// SIMATIC STEP 7 (V5.x) project CDCX52_Cordoba
// CPU: CPU
// station: P_ADR_BUS
// station: _S7H_BUSSYSTEM_CT
// station: Matériel
// station: API
// station: P_ADR_BUS
// station: Configuration
// station: MOP
// program: PROG
// program: Programa S7_BACK

SYMBOL_TABLE
"IBD"	DB 95	DB 95	// FACILITY: DATA BASE DB / DB BASE DE DONNEE
"IIT"	DB 96	DB 96	// FACILITY: PART TABLE / DB TABLE PIECE
"IIS"	DB 97	DB 97	// FACILITY: SUPPORT WORD TABLE / DB MOTS SUPPORT
"IG"	DB 99	DB 99	// FACILITY: GLOBAL DB / DB GLOBAL
END_SYMBOL_TABLE

DATA_BLOCK "IBD"	// DB 95
TITLE = FACILITY: DATABASE DB CONTROL
NAME : IBD
VERSION : 0.1
  STRUCT
   BDD : ARRAY  [1 .. 6, 1 .. 210 ] OF WORD ;	//SPARE
  END_STRUCT ;	
BEGIN
END_DATA_BLOCK

DATA_BLOCK "IIT"	// DB 96
TITLE = FACILITY: PART WORD TABLE
NAME : IIT
VERSION : 1.0
  STRUCT
   A01 : STRUCT 	//PALABRA PIEZA A01
    MP : STRUCT 	//PART MEMORY / PALABRA PIEZA
     MPP : BOOL ;	//PRESENT PART MEMORY / MEMORIA PIEZA PRESENTE
     MPAT : BOOL ;	//PART WITH WORK MEMORY / MEMORIA PIEZA A TRABAJAR
     MPST : BOOL ;	//PART WITHOUT WORK MEMORY / MEMORIA PIEZA SIN TRABAJO
     MPAM : BOOL ;	//PART MEMORY TO MATCH / MEMORIA PIEZA A CASAR
     MPAE : BOOL ;	//PART MEMORY TO EVACUATE / MEMORIA PIEZA A EVACUAR
     MPP1 : BOOL ;	//INTERMEDIATE PRESENT PART MEMORY / MEMORIA PIEZA PRESENTE INTERMEDIA
     MPP2 : BOOL ;	//INTERMEDIATE PRESENT PART MEMORY / MEMORIA PIEZA PRESENTE INTERMEDIA
     MPP3 : BOOL ;	//INTERMEDIATE PRESENT PART MEMORY / MEMORIA PIEZA PRESENTE INTERMEDIA
     MPP4 : BOOL ;	//INTERMEDIATE PRESENT PART MEMORY / MEMORIA PIEZA PRESENTE INTERMEDIA
     MPP5 : BOOL ;	//INTERMEDIATE PRESENT PART MEMORY / MEMORIA PIEZA PRESENTE INTERMEDIA
     MPP6 : BOOL ;	//INTERMEDIATE PRESENT PART MEMORY / MEMORIA PIEZA PRESENTE INTERMEDIA
     MPP7 : BOOL ;	//INTERMEDIATE PRESENT PART MEMORY / MEMORIA PIEZA PRESENTE INTERMEDIA
     MPP8 : BOOL ;	//INTERMEDIATE PRESENT PART MEMORY / MEMORIA PIEZA PRESENTE INTERMEDIA
     MPT : BOOL ;	//PART COMPLETE MEMORY / MEMORIA PIEZA TRABAJADA
     MPLNOK : BOOL ;	//LAUCHING PART MEMORY NOK / MEMORIA LANZAMIENTO PIEZA NO OK
     MPLNOR : BOOL ;	//LAUCHING PART MEMORY OK / MEMORIA LANZAMIENTO PIEZA OK
    END_STRUCT ;
    MS : INT ;
    NFILM : INT ;	//FILM NUMBER / NUMERO DE FILMO
    NORDRE : INT ;	//ORDER NUMBER / NUMERO DE ORDEN
    CDIV1 : INT ;	//FAMILIA (CDIV1)
    CDIV2 : INT ;	//FASE (CDIV2)
    CDIV3 : INT ;	//MODELO (CDIV3)
    CDIV4 : INT ;	//TECHO (CDIV4)
    CDIV5 : INT ;	//VERSION (CDIV5)
    DESFI : INT ;	//FINAL DISPATCH / DESTINO FINAL
    CSORT : INT ;	//TRADUCTION / CAUSA DE SALIDA
    DAT : STRUCT 	//DEFINICION / ESPERA TRABAJO
     B8 : BOOL ;
     B9 : BOOL ;
     B10 : BOOL ;
     B11 : BOOL ;
     B12 : BOOL ;
     FABSPF : BOOL ;	//FABRICACION SIN PIEZA AL FILMO
     B14 : BOOL ;
     B15 : BOOL ;
     B0 : BOOL ;
     B1 : BOOL ;
     B2 : BOOL ;
     B3 : BOOL ;
     B4 : BOOL ;
     B5 : BOOL ;
     B6 : BOOL ;
     B7 : BOOL ;
    END_STRUCT ;
    CRAPI : STRUCT 	//PLC DISPATCHING REASON / CAUSA ENRUTADO API
     B8 : BOOL ;
     B9 : BOOL ;
     B10 : BOOL ;
     B11 : BOOL ;
     B12 : BOOL ;
     B13 : BOOL ;
     B14 : BOOL ;
     B15 : BOOL ;
     B0 : BOOL ;
     B1 : BOOL ;
     B2 : BOOL ;
     RARET : BOOL ;	//PIEZA ANALISIS - RETOQUE
     B4 : BOOL ;
     B5 : BOOL ;
     B6 : BOOL ;
     B7 : BOOL ;
    END_STRUCT ;
    MGEST : STRUCT 	//PALABRA DE GESTION RECALAJE
     MPFNOR : BOOL ;	//MEMORIA PIEZA FLUJO NORMAL
     MPSTC : BOOL ;	//MEMORIA PIEZA A SALIR TODOS LOS CASOS
     MPSOR : BOOL ;	//MEMORIA PIEZA A SALIR (SALIDA SIPTOL BUENA)
     MPSSU : BOOL ;	//MEMORIA PIEZA A SALIR (SUSTITUCION PIEZA BUENA)
     MPSDI : BOOL ;	//MEMORIA PIEZA A SALIR (DISCORDANCIA)
     MPSSUL : BOOL ;	//MEMORIA PIEZA A SALIR (SUSTITUCION PIEZA MALA)
     MPSL : BOOL ;	//MEMORIA PIEZA A SALIR (SALIDA MALA)
     MPSF99 : BOOL ;	//MEMORIA PIEZA A SALIR (MAP FILM 99)
     MPETC : BOOL ;	//MEMORIA PIEZA A ENTRAR TODOS LOS CASOS
     MPEOR : BOOL ;	//MEMORIA PIEZA EN ENTRADA (DEMANDA SIPTOL)
     MPESUB : BOOL ;	//MEMORIA PIEZA EN ENTRADA (SUSTITUCION PIEZA BUENA)
     MPEDI : BOOL ;	//MEMORIA PIEZA EN ENTRADA (DISCORDANCIA)
     MPESUL : BOOL ;	//MEMORIA PIEZA EN ENTRADA (SUSTITUCION PIEZA MALA)
     MPOCV : BOOL ;	//MEMORIA PIEZA A SALIR VEHICULO ANULADO + GANCHO VACIO
     MESUTC : BOOL ;	//MEMORIA EN ENTRADA SUSTITUCION TODOS LOS CASOS (PIEZA BUENA O MALA)
     MSSUTC : BOOL ;	//MEMORIA SALIDA SUSTITUCION TODOS LOS CASOS (PIEZA BUENA O MALA)
    END_STRUCT ;
    TVEH : STRUCT 	//TYPO DE VEHICULO
     B8 : BOOL ;
     B9 : BOOL ;
     B10 : BOOL ;
     B11 : BOOL ;
     B12 : BOOL ;
     B13 : BOOL ;
     B14 : BOOL ;
     FABSPF : BOOL ;	//FABRICACION SIN PIEZA AL FILMO
     SPE : BOOL ;	//UNIT ESPECIAL
     B1 : BOOL ;
     B2 : BOOL ;
     B3 : BOOL ;
     B4 : BOOL ;
     B5 : BOOL ;
     B6 : BOOL ;
     B7 : BOOL ;
    END_STRUCT ;
    SPARE : ARRAY  [1 .. 5 ] OF INT ;	//SPARE
   END_STRUCT ;
   B01 : STRUCT 	//PALABRA PIEZA B01
    MP : STRUCT 	//PART MEMORY / PALABRA PIEZA
     MPP : BOOL ;	//PRESENT PART MEMORY / MEMORIA PIEZA PRESENTE
     MPAT : BOOL ;	//PART WITH WORK MEMORY / MEMORIA PIEZA A TRABAJAR
     MPST : BOOL ;	//PART WITHOUT WORK MEMORY / MEMORIA PIEZA SIN TRABAJO
     MPAM : BOOL ;	//PART MEMORY TO MATCH / MEMORIA PIEZA A CASAR
     MPAE : BOOL ;	//PART MEMORY TO EVACUATE / MEMORIA PIEZA A EVACUAR
     MPP1 : BOOL ;	//INTERMEDIATE PRESENT PART MEMORY / MEMORIA PIEZA PRESENTE INTERMEDIA
     MPP2 : BOOL ;	//INTERMEDIATE PRESENT PART MEMORY / MEMORIA PIEZA PRESENTE INTERMEDIA
     MPP3 : BOOL ;	//INTERMEDIATE PRESENT PART MEMORY / MEMORIA PIEZA PRESENTE INTERMEDIA
     MPP4 : BOOL ;	//INTERMEDIATE PRESENT PART MEMORY / MEMORIA PIEZA PRESENTE INTERMEDIA
     MPP5 : BOOL ;	//INTERMEDIATE PRESENT PART MEMORY / MEMORIA PIEZA PRESENTE INTERMEDIA
     MPP6 : BOOL ;	//INTERMEDIATE PRESENT PART MEMORY / MEMORIA PIEZA PRESENTE INTERMEDIA
     MPP7 : BOOL ;	//INTERMEDIATE PRESENT PART MEMORY / MEMORIA PIEZA PRESENTE INTERMEDIA
     MPP8 : BOOL ;	//INTERMEDIATE PRESENT PART MEMORY / MEMORIA PIEZA PRESENTE INTERMEDIA
     MPT : BOOL ;	//PART COMPLETE MEMORY / MEMORIA PIEZA TRABAJADA
     MPLNOK : BOOL ;	//LAUCHING PART MEMORY NOK / MEMORIA LANZAMIENTO PIEZA NO OK
     MPLNOR : BOOL ;	//LAUCHING PART MEMORY OK / MEMORIA LANZAMIENTO PIEZA OK
    END_STRUCT ;
    MS : INT ;
    NFILM : INT ;	//FILM NUMBER / NUMERO DE FILMO
    NORDRE : INT ;	//ORDER NUMBER / NUMERO DE ORDEN
    CDIV1 : INT ;	//FAMILIA (CDIV1)
    CDIV2 : INT ;	//FASE (CDIV2)
    CDIV3 : INT ;	//MODELO (CDIV3)
    CDIV4 : INT ;	//TECHO (CDIV4)
    CDIV5 : INT ;	//VERSION (CDIV5)
    DESFI : INT ;	//FINAL DISPATCH / DESTINO FINAL
    CSORT : INT ;	//TRADUCTION / CAUSA DE SALIDA
    DAT : STRUCT 	//DEFINICION / ESPERA TRABAJO
     B8 : BOOL ;
     B9 : BOOL ;
     B10 : BOOL ;
     B11 : BOOL ;
     B12 : BOOL ;
     FABSPF : BOOL ;	//FABRICACION SIN PIEZA AL FILMO
     B14 : BOOL ;
     B15 : BOOL ;
     B0 : BOOL ;
     B1 : BOOL ;
     B2 : BOOL ;
     B3 : BOOL ;
     B4 : BOOL ;
     B5 : BOOL ;
     B6 : BOOL ;
     B7 : BOOL ;
    END_STRUCT ;
    CRAPI : STRUCT 	//PLC DISPATCHING REASON / CAUSA ENRUTADO API
     B8 : BOOL ;
     B9 : BOOL ;
     B10 : BOOL ;
     B11 : BOOL ;
     B12 : BOOL ;
     B13 : BOOL ;
     B14 : BOOL ;
     B15 : BOOL ;
     B0 : BOOL ;
     B1 : BOOL ;
     B2 : BOOL ;
     RARET : BOOL ;	//PIEZA ANALISIS - RETOQUE
     B4 : BOOL ;
     B5 : BOOL ;
     B6 : BOOL ;
     B7 : BOOL ;
    END_STRUCT ;
    MGEST : STRUCT 	//PALABRA DE GESTION RECALAJE
     MPFNOR : BOOL ;	//MEMORIA PIEZA FLUJO NORMAL
     MPSTC : BOOL ;	//MEMORIA PIEZA A SALIR TODOS LOS CASOS
     MPSOR : BOOL ;	//MEMORIA PIEZA A SALIR (SALIDA SIPTOL BUENA)
     MPSSU : BOOL ;	//MEMORIA PIEZA A SALIR (SUSTITUCION PIEZA BUENA)
     MPSDI : BOOL ;	//MEMORIA PIEZA A SALIR (DISCORDANCIA)
     MPSSUL : BOOL ;	//MEMORIA PIEZA A SALIR (SUSTITUCION PIEZA MALA)
     MPSL : BOOL ;	//MEMORIA PIEZA A SALIR (SALIDA MALA)
     MPSF99 : BOOL ;	//MEMORIA PIEZA A SALIR (MAP FILM 99)
     MPETC : BOOL ;	//MEMORIA PIEZA A ENTRAR TODOS LOS CASOS
     MPEOR : BOOL ;	//MEMORIA PIEZA EN ENTRADA (DEMANDA SIPTOL)
     MPESUB : BOOL ;	//MEMORIA PIEZA EN ENTRADA (SUSTITUCION PIEZA BUENA)
     MPEDI : BOOL ;	//MEMORIA PIEZA EN ENTRADA (DISCORDANCIA)
     MPESUL : BOOL ;	//MEMORIA PIEZA EN ENTRADA (SUSTITUCION PIEZA MALA)
     MPOCV : BOOL ;	//MEMORIA PIEZA A SALIR VEHICULO ANULADO + GANCHO VACIO
     MESUTC : BOOL ;	//MEMORIA EN ENTRADA SUSTITUCION TODOS LOS CASOS (PIEZA BUENA O MALA)
     MSSUTC : BOOL ;	//MEMORIA SALIDA SUSTITUCION TODOS LOS CASOS (PIEZA BUENA O MALA)
    END_STRUCT ;
    TVEH : STRUCT 	//TYPO DE VEHICULO
     B8 : BOOL ;
     B9 : BOOL ;
     B10 : BOOL ;
     B11 : BOOL ;
     B12 : BOOL ;
     B13 : BOOL ;
     B14 : BOOL ;
     FABSPF : BOOL ;	//FABRICACION SIN PIEZA AL FILMO
     SPE : BOOL ;	//UNIT ESPECIAL
     B1 : BOOL ;
     B2 : BOOL ;
     B3 : BOOL ;
     B4 : BOOL ;
     B5 : BOOL ;
     B6 : BOOL ;
     B7 : BOOL ;
    END_STRUCT ;
    SPARE : ARRAY  [1 .. 5 ] OF INT ;
   END_STRUCT ;
   B02 : STRUCT 	//PALABRA PIEZA B02
    MP : STRUCT 	//PART MEMORY / PALABRA PIEZA
     MPP : BOOL ;	//PRESENT PART MEMORY / MEMORIA PIEZA PRESENTE
     MPAT : BOOL ;	//PART WITH WORK MEMORY / MEMORIA PIEZA A TRABAJAR
     MPST : BOOL ;	//PART WITHOUT WORK MEMORY / MEMORIA PIEZA SIN TRABAJO
     MPAM : BOOL ;	//PART MEMORY TO MATCH / MEMORIA PIEZA A CASAR
     MPAE : BOOL ;	//PART MEMORY TO EVACUATE / MEMORIA PIEZA A EVACUAR
     MPP1 : BOOL ;	//INTERMEDIATE PRESENT PART MEMORY / MEMORIA PIEZA PRESENTE INTERMEDIA
     MPP2 : BOOL ;	//INTERMEDIATE PRESENT PART MEMORY / MEMORIA PIEZA PRESENTE INTERMEDIA
     MPP3 : BOOL ;	//INTERMEDIATE PRESENT PART MEMORY / MEMORIA PIEZA PRESENTE INTERMEDIA
     MPP4 : BOOL ;	//INTERMEDIATE PRESENT PART MEMORY / MEMORIA PIEZA PRESENTE INTERMEDIA
     MPP5 : BOOL ;	//INTERMEDIATE PRESENT PART MEMORY / MEMORIA PIEZA PRESENTE INTERMEDIA
     MPP6 : BOOL ;	//INTERMEDIATE PRESENT PART MEMORY / MEMORIA PIEZA PRESENTE INTERMEDIA
     MPP7 : BOOL ;	//INTERMEDIATE PRESENT PART MEMORY / MEMORIA PIEZA PRESENTE INTERMEDIA
     MPP8 : BOOL ;	//INTERMEDIATE PRESENT PART MEMORY / MEMORIA PIEZA PRESENTE INTERMEDIA
     MPT : BOOL ;	//PART COMPLETE MEMORY / MEMORIA PIEZA TRABAJADA
     MPLNOK : BOOL ;	//LAUCHING PART MEMORY NOK / MEMORIA LANZAMIENTO PIEZA NO OK
     MPLNOR : BOOL ;	//LAUCHING PART MEMORY OK / MEMORIA LANZAMIENTO PIEZA OK
    END_STRUCT ;
    MS : INT ;
    NFILM : INT ;	//FILM NUMBER / NUMERO DE FILMO
    NORDRE : INT ;	//ORDER NUMBER / NUMERO DE ORDEN
    CDIV1 : INT ;	//FAMILIA (CDIV1)
    CDIV2 : INT ;	//FASE (CDIV2)
    CDIV3 : INT ;	//MODELO (CDIV3)
    CDIV4 : INT ;	//TECHO (CDIV4)
    CDIV5 : INT ;	//VERSION (CDIV5)
    DESFI : INT ;	//FINAL DISPATCH / DESTINO FINAL
    CSORT : INT ;	//TRADUCTION / CAUSA DE SALIDA
    DAT : STRUCT 	//DEFINICION / ESPERA TRABAJO
     B8 : BOOL ;
     B9 : BOOL ;
     B10 : BOOL ;
     B11 : BOOL ;
     B12 : BOOL ;
     FABSPF : BOOL ;	//FABRICACION SIN PIEZA AL FILMO
     B14 : BOOL ;
     B15 : BOOL ;
     B0 : BOOL ;
     B1 : BOOL ;
     B2 : BOOL ;
     B3 : BOOL ;
     B4 : BOOL ;
     B5 : BOOL ;
     B6 : BOOL ;
     B7 : BOOL ;
    END_STRUCT ;
    CRAPI : STRUCT 	//PLC DISPATCHING REASON / CAUSA ENRUTADO API
     B8 : BOOL ;
     B9 : BOOL ;
     B10 : BOOL ;
     B11 : BOOL ;
     B12 : BOOL ;
     B13 : BOOL ;
     B14 : BOOL ;
     B15 : BOOL ;
     B0 : BOOL ;
     B1 : BOOL ;
     B2 : BOOL ;
     RARET : BOOL ;	//PIEZA ANALISIS - RETOQUE
     B4 : BOOL ;
     B5 : BOOL ;
     B6 : BOOL ;
     B7 : BOOL ;
    END_STRUCT ;
    MGEST : STRUCT 	//PALABRA DE GESTION RECALAJE
     MPFNOR : BOOL ;	//MEMORIA PIEZA FLUJO NORMAL
     MPSTC : BOOL ;	//MEMORIA PIEZA A SALIR TODOS LOS CASOS
     MPSOR : BOOL ;	//MEMORIA PIEZA A SALIR (SALIDA SIPTOL BUENA)
     MPSSU : BOOL ;	//MEMORIA PIEZA A SALIR (SUSTITUCION PIEZA BUENA)
     MPSDI : BOOL ;	//MEMORIA PIEZA A SALIR (DISCORDANCIA)
     MPSSUL : BOOL ;	//MEMORIA PIEZA A SALIR (SUSTITUCION PIEZA MALA)
     MPSL : BOOL ;	//MEMORIA PIEZA A SALIR (SALIDA MALA)
     MPSF99 : BOOL ;	//MEMORIA PIEZA A SALIR (MAP FILM 99)
     MPETC : BOOL ;	//MEMORIA PIEZA A ENTRAR TODOS LOS CASOS
     MPEOR : BOOL ;	//MEMORIA PIEZA EN ENTRADA (DEMANDA SIPTOL)
     MPESUB : BOOL ;	//MEMORIA PIEZA EN ENTRADA (SUSTITUCION PIEZA BUENA)
     MPEDI : BOOL ;	//MEMORIA PIEZA EN ENTRADA (DISCORDANCIA)
     MPESUL : BOOL ;	//MEMORIA PIEZA EN ENTRADA (SUSTITUCION PIEZA MALA)
     MPOCV : BOOL ;	//MEMORIA PIEZA A SALIR VEHICULO ANULADO + GANCHO VACIO
     MESUTC : BOOL ;	//MEMORIA EN ENTRADA SUSTITUCION TODOS LOS CASOS (PIEZA BUENA O MALA)
     MSSUTC : BOOL ;	//MEMORIA SALIDA SUSTITUCION TODOS LOS CASOS (PIEZA BUENA O MALA)
    END_STRUCT ;
    TVEH : STRUCT 	//TYPO DE VEHICULO
     B8 : BOOL ;
     B9 : BOOL ;
     B10 : BOOL ;
     B11 : BOOL ;
     B12 : BOOL ;
     B13 : BOOL ;
     B14 : BOOL ;
     FABSPF : BOOL ;	//FABRICACION SIN PIEZA AL FILMO
     SPE : BOOL ;	//UNIT ESPECIAL
     B1 : BOOL ;
     B2 : BOOL ;
     B3 : BOOL ;
     B4 : BOOL ;
     B5 : BOOL ;
     B6 : BOOL ;
     B7 : BOOL ;
    END_STRUCT ;
    SPARE : ARRAY  [1 .. 5 ] OF INT ;
   END_STRUCT ;
   C01 : STRUCT 	//PALABRA PIEZA C01
    MP : STRUCT 	//PART MEMORY / PALABRA PIEZA
     MPP : BOOL ;	//PRESENT PART MEMORY / MEMORIA PIEZA PRESENTE
     MPAT : BOOL ;	//PART WITH WORK MEMORY / MEMORIA PIEZA A TRABAJAR
     MPST : BOOL ;	//PART WITHOUT WORK MEMORY / MEMORIA PIEZA SIN TRABAJO
     MPAM : BOOL ;	//PART MEMORY TO MATCH / MEMORIA PIEZA A CASAR
     MPAE : BOOL ;	//PART MEMORY TO EVACUATE / MEMORIA PIEZA A EVACUAR
     MPP1 : BOOL ;	//INTERMEDIATE PRESENT PART MEMORY / MEMORIA PIEZA PRESENTE INTERMEDIA
     MPP2 : BOOL ;	//INTERMEDIATE PRESENT PART MEMORY / MEMORIA PIEZA PRESENTE INTERMEDIA
     MPP3 : BOOL ;	//INTERMEDIATE PRESENT PART MEMORY / MEMORIA PIEZA PRESENTE INTERMEDIA
     MPP4 : BOOL ;	//INTERMEDIATE PRESENT PART MEMORY / MEMORIA PIEZA PRESENTE INTERMEDIA
     MPP5 : BOOL ;	//INTERMEDIATE PRESENT PART MEMORY / MEMORIA PIEZA PRESENTE INTERMEDIA
     MPP6 : BOOL ;	//INTERMEDIATE PRESENT PART MEMORY / MEMORIA PIEZA PRESENTE INTERMEDIA
     MPP7 : BOOL ;	//INTERMEDIATE PRESENT PART MEMORY / MEMORIA PIEZA PRESENTE INTERMEDIA
     MPP8 : BOOL ;	//INTERMEDIATE PRESENT PART MEMORY / MEMORIA PIEZA PRESENTE INTERMEDIA
     MPT : BOOL ;	//PART COMPLETE MEMORY / MEMORIA PIEZA TRABAJADA
     MPLNOK : BOOL ;	//LAUCHING PART MEMORY NOK / MEMORIA LANZAMIENTO PIEZA NO OK
     MPLNOR : BOOL ;	//LAUCHING PART MEMORY OK / MEMORIA LANZAMIENTO PIEZA OK
    END_STRUCT ;
    MS : INT ;
    NFILM : INT ;	//FILM NUMBER / NUMERO DE FILMO
    NORDRE : INT ;	//ORDER NUMBER / NUMERO DE ORDEN
    CDIV1 : INT ;	//FAMILIA (CDIV1)
    CDIV2 : INT ;	//FASE (CDIV2)
    CDIV3 : INT ;	//MODELO (CDIV3)
    CDIV4 : INT ;	//TECHO (CDIV4)
    CDIV5 : INT ;	//VERSION (CDIV5)
    DESFI : INT ;	//FINAL DISPATCH / DESTINO FINAL
    CSORT : INT ;	//TRADUCTION / CAUSA DE SALIDA
    DAT : STRUCT 	//DEFINICION / ESPERA TRABAJO
     B8 : BOOL ;
     B9 : BOOL ;
     B10 : BOOL ;
     B11 : BOOL ;
     B12 : BOOL ;
     FABSPF : BOOL ;	//FABRICACION SIN PIEZA AL FILMO
     B14 : BOOL ;
     B15 : BOOL ;
     B0 : BOOL ;
     B1 : BOOL ;
     B2 : BOOL ;
     B3 : BOOL ;
     B4 : BOOL ;
     B5 : BOOL ;
     B6 : BOOL ;
     B7 : BOOL ;
    END_STRUCT ;
    CRAPI : STRUCT 	//PLC DISPATCHING REASON / CAUSA ENRUTADO API
     B8 : BOOL ;
     B9 : BOOL ;
     B10 : BOOL ;
     B11 : BOOL ;
     B12 : BOOL ;
     B13 : BOOL ;
     B14 : BOOL ;
     B15 : BOOL ;
     B0 : BOOL ;
     B1 : BOOL ;
     B2 : BOOL ;
     RARET : BOOL ;	//PIEZA ANALISIS - RETOQUE
     B4 : BOOL ;
     B5 : BOOL ;
     B6 : BOOL ;
     B7 : BOOL ;
    END_STRUCT ;
    MGEST : STRUCT 	//PALABRA DE GESTION RECALAJE
     MPFNOR : BOOL ;	//MEMORIA PIEZA FLUJO NORMAL
     MPSTC : BOOL ;	//MEMORIA PIEZA A SALIR TODOS LOS CASOS
     MPSOR : BOOL ;	//MEMORIA PIEZA A SALIR (SALIDA SIPTOL BUENA)
     MPSSU : BOOL ;	//MEMORIA PIEZA A SALIR (SUSTITUCION PIEZA BUENA)
     MPSDI : BOOL ;	//MEMORIA PIEZA A SALIR (DISCORDANCIA)
     MPSSUL : BOOL ;	//MEMORIA PIEZA A SALIR (SUSTITUCION PIEZA MALA)
     MPSL : BOOL ;	//MEMORIA PIEZA A SALIR (SALIDA MALA)
     MPSF99 : BOOL ;	//MEMORIA PIEZA A SALIR (MAP FILM 99)
     MPETC : BOOL ;	//MEMORIA PIEZA A ENTRAR TODOS LOS CASOS
     MPEOR : BOOL ;	//MEMORIA PIEZA EN ENTRADA (DEMANDA SIPTOL)
     MPESUB : BOOL ;	//MEMORIA PIEZA EN ENTRADA (SUSTITUCION PIEZA BUENA)
     MPEDI : BOOL ;	//MEMORIA PIEZA EN ENTRADA (DISCORDANCIA)
     MPESUL : BOOL ;	//MEMORIA PIEZA EN ENTRADA (SUSTITUCION PIEZA MALA)
     MPOCV : BOOL ;	//MEMORIA PIEZA A SALIR VEHICULO ANULADO + GANCHO VACIO
     MESUTC : BOOL ;	//MEMORIA EN ENTRADA SUSTITUCION TODOS LOS CASOS (PIEZA BUENA O MALA)
     MSSUTC : BOOL ;	//MEMORIA SALIDA SUSTITUCION TODOS LOS CASOS (PIEZA BUENA O MALA)
    END_STRUCT ;
    TVEH : STRUCT 	//TYPO DE VEHICULO
     B8 : BOOL ;
     B9 : BOOL ;
     B10 : BOOL ;
     B11 : BOOL ;
     B12 : BOOL ;
     B13 : BOOL ;
     B14 : BOOL ;
     FABSPF : BOOL ;	//FABRICACION SIN PIEZA AL FILMO
     SPE : BOOL ;	//UNIT ESPECIAL
     B1 : BOOL ;
     B2 : BOOL ;
     B3 : BOOL ;
     B4 : BOOL ;
     B5 : BOOL ;
     B6 : BOOL ;
     B7 : BOOL ;
    END_STRUCT ;
    SPARE : ARRAY  [1 .. 5 ] OF INT ;
   END_STRUCT ;
   C02 : STRUCT 	//PALABRA PIEZA C02
    MP : STRUCT 	//PART MEMORY / PALABRA PIEZA
     MPP : BOOL ;	//PRESENT PART MEMORY / MEMORIA PIEZA PRESENTE
     MPAT : BOOL ;	//PART WITH WORK MEMORY / MEMORIA PIEZA A TRABAJAR
     MPST : BOOL ;	//PART WITHOUT WORK MEMORY / MEMORIA PIEZA SIN TRABAJO
     MPAM : BOOL ;	//PART MEMORY TO MATCH / MEMORIA PIEZA A CASAR
     MPAE : BOOL ;	//PART MEMORY TO EVACUATE / MEMORIA PIEZA A EVACUAR
     MPP1 : BOOL ;	//INTERMEDIATE PRESENT PART MEMORY / MEMORIA PIEZA PRESENTE INTERMEDIA
     MPP2 : BOOL ;	//INTERMEDIATE PRESENT PART MEMORY / MEMORIA PIEZA PRESENTE INTERMEDIA
     MPP3 : BOOL ;	//INTERMEDIATE PRESENT PART MEMORY / MEMORIA PIEZA PRESENTE INTERMEDIA
     MPP4 : BOOL ;	//INTERMEDIATE PRESENT PART MEMORY / MEMORIA PIEZA PRESENTE INTERMEDIA
     MPP5 : BOOL ;	//INTERMEDIATE PRESENT PART MEMORY / MEMORIA PIEZA PRESENTE INTERMEDIA
     MPP6 : BOOL ;	//INTERMEDIATE PRESENT PART MEMORY / MEMORIA PIEZA PRESENTE INTERMEDIA
     MPP7 : BOOL ;	//INTERMEDIATE PRESENT PART MEMORY / MEMORIA PIEZA PRESENTE INTERMEDIA
     MPP8 : BOOL ;	//INTERMEDIATE PRESENT PART MEMORY / MEMORIA PIEZA PRESENTE INTERMEDIA
     MPT : BOOL ;	//PART COMPLETE MEMORY / MEMORIA PIEZA TRABAJADA
     MPLNOK : BOOL ;	//LAUCHING PART MEMORY NOK / MEMORIA LANZAMIENTO PIEZA NO OK
     MPLNOR : BOOL ;	//LAUCHING PART MEMORY OK / MEMORIA LANZAMIENTO PIEZA OK
    END_STRUCT ;
    MS : INT ;
    NFILM : INT ;	//FILM NUMBER / NUMERO DE FILMO
    NORDRE : INT ;	//ORDER NUMBER / NUMERO DE ORDEN
    CDIV1 : INT ;	//FAMILIA (CDIV1)
    CDIV2 : INT ;	//FASE (CDIV2)
    CDIV3 : INT ;	//MODELO (CDIV3)
    CDIV4 : INT ;	//TECHO (CDIV4)
    CDIV5 : INT ;	//VERSION (CDIV5)
    DESFI : INT ;	//FINAL DISPATCH / DESTINO FINAL
    CSORT : INT ;	//TRADUCTION / CAUSA DE SALIDA
    DAT : STRUCT 	//DEFINICION / ESPERA TRABAJO
     B8 : BOOL ;
     B9 : BOOL ;
     B10 : BOOL ;
     B11 : BOOL ;
     B12 : BOOL ;
     FABSPF : BOOL ;	//FABRICACION SIN PIEZA AL FILMO
     B14 : BOOL ;
     B15 : BOOL ;
     B0 : BOOL ;
     B1 : BOOL ;
     B2 : BOOL ;
     B3 : BOOL ;
     B4 : BOOL ;
     B5 : BOOL ;
     B6 : BOOL ;
     B7 : BOOL ;
    END_STRUCT ;
    CRAPI : STRUCT 	//PLC DISPATCHING REASON / CAUSA ENRUTADO API
     B8 : BOOL ;
     B9 : BOOL ;
     B10 : BOOL ;
     B11 : BOOL ;
     B12 : BOOL ;
     B13 : BOOL ;
     B14 : BOOL ;
     B15 : BOOL ;
     B0 : BOOL ;
     B1 : BOOL ;
     B2 : BOOL ;
     RARET : BOOL ;	//PIEZA ANALISIS - RETOQUE
     B4 : BOOL ;
     B5 : BOOL ;
     B6 : BOOL ;
     B7 : BOOL ;
    END_STRUCT ;
    MGEST : STRUCT 	//PALABRA DE GESTION RECALAJE
     MPFNOR : BOOL ;	//MEMORIA PIEZA FLUJO NORMAL
     MPSTC : BOOL ;	//MEMORIA PIEZA A SALIR TODOS LOS CASOS
     MPSOR : BOOL ;	//MEMORIA PIEZA A SALIR (SALIDA SIPTOL BUENA)
     MPSSU : BOOL ;	//MEMORIA PIEZA A SALIR (SUSTITUCION PIEZA BUENA)
     MPSDI : BOOL ;	//MEMORIA PIEZA A SALIR (DISCORDANCIA)
     MPSSUL : BOOL ;	//MEMORIA PIEZA A SALIR (SUSTITUCION PIEZA MALA)
     MPSL : BOOL ;	//MEMORIA PIEZA A SALIR (SALIDA MALA)
     MPSF99 : BOOL ;	//MEMORIA PIEZA A SALIR (MAP FILM 99)
     MPETC : BOOL ;	//MEMORIA PIEZA A ENTRAR TODOS LOS CASOS
     MPEOR : BOOL ;	//MEMORIA PIEZA EN ENTRADA (DEMANDA SIPTOL)
     MPESUB : BOOL ;	//MEMORIA PIEZA EN ENTRADA (SUSTITUCION PIEZA BUENA)
     MPEDI : BOOL ;	//MEMORIA PIEZA EN ENTRADA (DISCORDANCIA)
     MPESUL : BOOL ;	//MEMORIA PIEZA EN ENTRADA (SUSTITUCION PIEZA MALA)
     MPOCV : BOOL ;	//MEMORIA PIEZA A SALIR VEHICULO ANULADO + GANCHO VACIO
     MESUTC : BOOL ;	//MEMORIA EN ENTRADA SUSTITUCION TODOS LOS CASOS (PIEZA BUENA O MALA)
     MSSUTC : BOOL ;	//MEMORIA SALIDA SUSTITUCION TODOS LOS CASOS (PIEZA BUENA O MALA)
    END_STRUCT ;
    TVEH : STRUCT 	//TYPO DE VEHICULO
     B8 : BOOL ;
     B9 : BOOL ;
     B10 : BOOL ;
     B11 : BOOL ;
     B12 : BOOL ;
     B13 : BOOL ;
     B14 : BOOL ;
     FABSPF : BOOL ;	//FABRICACION SIN PIEZA AL FILMO
     SPE : BOOL ;	//UNIT ESPECIAL
     B1 : BOOL ;
     B2 : BOOL ;
     B3 : BOOL ;
     B4 : BOOL ;
     B5 : BOOL ;
     B6 : BOOL ;
     B7 : BOOL ;
    END_STRUCT ;
    SPARE : ARRAY  [1 .. 5 ] OF INT ;
   END_STRUCT ;
   A01w : STRUCT 	//PALABRA PIEZA A01 transito
    MP : STRUCT 	//PART MEMORY / PALABRA PIEZA
     MPP : BOOL ;	//PRESENT PART MEMORY / MEMORIA PIEZA PRESENTE
     MPAT : BOOL ;	//PART WITH WORK MEMORY / MEMORIA PIEZA A TRABAJAR
     MPST : BOOL ;	//PART WITHOUT WORK MEMORY / MEMORIA PIEZA SIN TRABAJO
     MPAM : BOOL ;	//PART MEMORY TO MATCH / MEMORIA PIEZA A CASAR
     MPAE : BOOL ;	//PART MEMORY TO EVACUATE / MEMORIA PIEZA A EVACUAR
     MPP1 : BOOL ;	//INTERMEDIATE PRESENT PART MEMORY / MEMORIA PIEZA PRESENTE INTERMEDIA
     MPP2 : BOOL ;	//INTERMEDIATE PRESENT PART MEMORY / MEMORIA PIEZA PRESENTE INTERMEDIA
     MPP3 : BOOL ;	//INTERMEDIATE PRESENT PART MEMORY / MEMORIA PIEZA PRESENTE INTERMEDIA
     MPP4 : BOOL ;	//INTERMEDIATE PRESENT PART MEMORY / MEMORIA PIEZA PRESENTE INTERMEDIA
     MPP5 : BOOL ;	//INTERMEDIATE PRESENT PART MEMORY / MEMORIA PIEZA PRESENTE INTERMEDIA
     MPP6 : BOOL ;	//INTERMEDIATE PRESENT PART MEMORY / MEMORIA PIEZA PRESENTE INTERMEDIA
     MPP7 : BOOL ;	//INTERMEDIATE PRESENT PART MEMORY / MEMORIA PIEZA PRESENTE INTERMEDIA
     MPP8 : BOOL ;	//INTERMEDIATE PRESENT PART MEMORY / MEMORIA PIEZA PRESENTE INTERMEDIA
     MPT : BOOL ;	//PART COMPLETE MEMORY / MEMORIA PIEZA TRABAJADA
     MPLNOK : BOOL ;	//LAUCHING PART MEMORY NOK / MEMORIA LANZAMIENTO PIEZA NO OK
     MPLNOR : BOOL ;	//LAUCHING PART MEMORY OK / MEMORIA LANZAMIENTO PIEZA OK
    END_STRUCT ;
    MS : INT ;
    NFILM : INT ;	//FILM NUMBER / NUMERO DE FILMO
    NORDRE : INT ;	//ORDER NUMBER / NUMERO DE ORDEN
    CDIV1 : INT ;	//FAMILIA (CDIV1)
    CDIV2 : INT ;	//FASE (CDIV2)
    CDIV3 : INT ;	//MODELO (CDIV3)
    CDIV4 : INT ;	//TECHO (CDIV4)
    CDIV5 : INT ;	//VERSION (CDIV5)
    DESFI : INT ;	//FINAL DISPATCH / DESTINO FINAL
    CSORT : INT ;	//TRADUCTION / CAUSA DE SALIDA
    DAT : STRUCT 	//DEFINICION / ESPERA TRABAJO
     B8 : BOOL ;
     B9 : BOOL ;
     B10 : BOOL ;
     B11 : BOOL ;
     B12 : BOOL ;
     FABSPF : BOOL ;	//FABRICACION SIN PIEZA AL FILMO
     B14 : BOOL ;
     B15 : BOOL ;
     B0 : BOOL ;
     B1 : BOOL ;
     B2 : BOOL ;
     B3 : BOOL ;
     B4 : BOOL ;
     B5 : BOOL ;
     B6 : BOOL ;
     B7 : BOOL ;
    END_STRUCT ;
    CRAPI : STRUCT 	//PLC DISPATCHING REASON / CAUSA ENRUTADO API
     B8 : BOOL ;
     B9 : BOOL ;
     B10 : BOOL ;
     B11 : BOOL ;
     B12 : BOOL ;
     B13 : BOOL ;
     B14 : BOOL ;
     B15 : BOOL ;
     B0 : BOOL ;
     B1 : BOOL ;
     B2 : BOOL ;
     RARET : BOOL ;	//PIEZA ANALISIS - RETOQUE
     B4 : BOOL ;
     B5 : BOOL ;
     B6 : BOOL ;
     B7 : BOOL ;
    END_STRUCT ;
    MGEST : STRUCT 	//PALABRA DE GESTION RECALAJE
     MPFNOR : BOOL ;	//MEMORIA PIEZA FLUJO NORMAL
     MPSTC : BOOL ;	//MEMORIA PIEZA A SALIR TODOS LOS CASOS
     MPSOR : BOOL ;	//MEMORIA PIEZA A SALIR (SALIDA SIPTOL BUENA)
     MPSSU : BOOL ;	//MEMORIA PIEZA A SALIR (SUSTITUCION PIEZA BUENA)
     MPSDI : BOOL ;	//MEMORIA PIEZA A SALIR (DISCORDANCIA)
     MPSSUL : BOOL ;	//MEMORIA PIEZA A SALIR (SUSTITUCION PIEZA MALA)
     MPSL : BOOL ;	//MEMORIA PIEZA A SALIR (SALIDA MALA)
     MPSF99 : BOOL ;	//MEMORIA PIEZA A SALIR (MAP FILM 99)
     MPETC : BOOL ;	//MEMORIA PIEZA A ENTRAR TODOS LOS CASOS
     MPEOR : BOOL ;	//MEMORIA PIEZA EN ENTRADA (DEMANDA SIPTOL)
     MPESUB : BOOL ;	//MEMORIA PIEZA EN ENTRADA (SUSTITUCION PIEZA BUENA)
     MPEDI : BOOL ;	//MEMORIA PIEZA EN ENTRADA (DISCORDANCIA)
     MPESUL : BOOL ;	//MEMORIA PIEZA EN ENTRADA (SUSTITUCION PIEZA MALA)
     MPOCV : BOOL ;	//MEMORIA PIEZA A SALIR VEHICULO ANULADO + GANCHO VACIO
     MESUTC : BOOL ;	//MEMORIA EN ENTRADA SUSTITUCION TODOS LOS CASOS (PIEZA BUENA O MALA)
     MSSUTC : BOOL ;	//MEMORIA SALIDA SUSTITUCION TODOS LOS CASOS (PIEZA BUENA O MALA)
    END_STRUCT ;
    TVEH : STRUCT 	//TYPO DE VEHICULO
     B8 : BOOL ;
     B9 : BOOL ;
     B10 : BOOL ;
     B11 : BOOL ;
     B12 : BOOL ;
     B13 : BOOL ;
     B14 : BOOL ;
     FABSPF : BOOL ;	//FABRICACION SIN PIEZA AL FILMO
     SPE : BOOL ;	//UNIT ESPECIAL
     B1 : BOOL ;
     B2 : BOOL ;
     B3 : BOOL ;
     B4 : BOOL ;
     B5 : BOOL ;
     B6 : BOOL ;
     B7 : BOOL ;
    END_STRUCT ;
    SPARE : ARRAY  [1 .. 5 ] OF INT ;
   END_STRUCT ;
  END_STRUCT ;	
BEGIN
END_DATA_BLOCK

DATA_BLOCK "IIS"	// DB 97
TITLE = FACILITY: SUPPORT WORD TABLE / DB MOTS SUPPORT
VERSION : 0.1
  STRUCT
   K0C_1 : STRUCT 	//K0C_TOPE 1 : SUPPORT MEMORY / MEMORIA SOPORTE
    MSP : BOOL ;	//SUPPORT PRESENCIA MEMORY / MEMORIA SOPORTE PRESENTE
    MSE : BOOL ;	//SUPPORT EVACUATED MEMORY / MEMORIA SOPORTE EVACUADO
    MTE1 : BOOL ;	//WORK 1 COMPLETE MEMORY / MEMORIA TRABAJO 1 REALIZADO
    MTE2 : BOOL ;	//WORK 2 COMPLETE MEMORY / MEMORIA TRABAJO 2 REALIZADO
    MTE3 : BOOL ;	//WORK 3 COMPLETE MEMORY / MEMORIA TRABAJO 3 REALIZADO
    MS5 : BOOL ;	//SPARE / RESERVA
    MS6 : BOOL ;	//SPARE / RESERVA
    MSAE : BOOL ;	//SUPPORT TO EVACUATE MEMORY / MEMORIA SOPORTE A EVACUAR
    MSVIDE : BOOL ;	//SUPPORT EMPTY MEMORY / MEMORIA SOPORTE VACIO
    MSLRFID : BOOL ;	//SUPPORT MEMORY RFID READING OK / MEMORIA SOPORTE LECTURA RFID OK
    MSERFID : BOOL ;	//SUPPORT MEMORY RFID WRITING OK / MEMORIA SOPORTE ESCRITURA RFID OK
    MS11 : BOOL ;	//SPARE / RESERVA
    MS12 : BOOL ;	//SPARE / RESERVA
    MS13 : BOOL ;	//SPARE / RESERVA
    MS14 : BOOL ;	//SPARE / RESERVA
    MS15 : BOOL ;	//SPARE / RESERVA
   END_STRUCT ;
   K0C_2 : STRUCT 	//K0C_TOPE 2 : SUPPORT MEMORY / MEMORIA SOPORTE
    MSP : BOOL ;	//SUPPORT PRESENCIA MEMORY / MEMORIA SOPORTE PRESENTE
    MSE : BOOL ;	//SUPPORT EVACUATED MEMORY / MEMORIA SOPORTE EVACUADO
    MTE1 : BOOL ;	//WORK 1 COMPLETE MEMORY / MEMORIA TRABAJO 1 REALIZADO
    MTE2 : BOOL ;	//WORK 2 COMPLETE MEMORY / MEMORIA TRABAJO 2 REALIZADO
    MTE3 : BOOL ;	//WORK 3 COMPLETE MEMORY / MEMORIA TRABAJO 3 REALIZADO
    MS5 : BOOL ;	//SPARE / RESERVA
    MS6 : BOOL ;	//SPARE / RESERVA
    MSAE : BOOL ;	//SUPPORT TO EVACUATE MEMORY / MEMORIA SOPORTE A EVACUAR
    MSVIDE : BOOL ;	//SUPPORT EMPTY MEMORY / MEMORIA SOPORTE VACIO
    MSLRFID : BOOL ;	//SUPPORT MEMORY RFID READING OK / MEMORIA SOPORTE LECTURA RFID OK
    MSERFID : BOOL ;	//SUPPORT MEMORY RFID WRITING OK / MEMORIA SOPORTE ESCRITURA RFID OK
    MS11 : BOOL ;	//SPARE / RESERVA
    MS12 : BOOL ;	//SPARE / RESERVA
    MS13 : BOOL ;	//SPARE / RESERVA
    MS14 : BOOL ;	//SPARE / RESERVA
    MS15 : BOOL ;	//SPARE / RESERVA
   END_STRUCT ;
   F1 : STRUCT 	//F1 : SUPPORT MEMORY / MEMORIA SOPORTE
    MSP : BOOL ;	//SUPPORT PRESENCIA MEMORY / MEMORIA SOPORTE PRESENTE
    MS1 : BOOL ;	//SPARE / RESERVA
    MS2 : BOOL ;	//SPARE / RESERVA
    MS3 : BOOL ;	//SPARE / RESERVA
    MS4 : BOOL ;	//SPARE / RESERVA
    MS5 : BOOL ;	//SPARE / RESERVA
    MS6 : BOOL ;	//SPARE / RESERVA
    MS7 : BOOL ;	//SPARE / RESERVA
    MS8 : BOOL ;	//SPARE / RESERVA
    MS9 : BOOL ;	//SPARE / RESERVA
    MS10 : BOOL ;	//SPARE / RESERVA
    MS11 : BOOL ;	//SPARE / RESERVA
    MS12 : BOOL ;	//SPARE / RESERVA
    MS13 : BOOL ;	//SPARE / RESERVA
    MS14 : BOOL ;	//SPARE / RESERVA
    MS15 : BOOL ;	//SPARE / RESERVA
   END_STRUCT ;
   F2 : STRUCT 	//F2 : SUPPORT MEMORY / MEMORIA SOPORTE
    MSP : BOOL ;	//SUPPORT PRESENCIA MEMORY / MEMORIA SOPORTE PRESENTE
    MS1 : BOOL ;	//SPARE / RESERVA
    MS2 : BOOL ;	//SPARE / RESERVA
    MS3 : BOOL ;	//SPARE / RESERVA
    MS4 : BOOL ;	//SPARE / RESERVA
    MS5 : BOOL ;	//SPARE / RESERVA
    MS6 : BOOL ;	//SPARE / RESERVA
    MS7 : BOOL ;	//SPARE / RESERVA
    MS8 : BOOL ;	//SPARE / RESERVA
    MS9 : BOOL ;	//SPARE / RESERVA
    MS10 : BOOL ;	//SPARE / RESERVA
    MS11 : BOOL ;	//SPARE / RESERVA
    MS12 : BOOL ;	//SPARE / RESERVA
    MS13 : BOOL ;	//SPARE / RESERVA
    MS14 : BOOL ;	//SPARE / RESERVA
    MS15 : BOOL ;	//SPARE / RESERVA
   END_STRUCT ;
  END_STRUCT ;	
BEGIN
END_DATA_BLOCK

DATA_BLOCK "IG"	// DB 99
TITLE = FACILITY: GLOBAL DB
NAME : IG
VERSION : 0.1
  STRUCT
   VALEUR0 : BYTE ;	//BYTE ALWAYS OFF (SFC20) / OCTETO SIEMPRE A 0
   MAFJ : BOOL ;	//MEMORY STOP END DAY
   LIEN_ILOT : UDT 2004;	//FACILITY LINK / ENLACE ISLA
   DEF_MAJ : BOOL ;	//FACILITY: MAJOR FAULT / ISLA DEFECTO MAYOR
   WVALEUR0 : INT ;	//PALABRA SIEMPRE A 0
   MPVALEUR0 : ARRAY  [1 .. 20 ] OF //PALABRA PIEZA SIEMPRE A 0
   INT ;
   ITLG : BOOL ;	//FACILITY: GENERAL LAMP TEST INFORMATION / INFO TEST LAMPE GENERAL
   ICL : BOOL ;	//FACILITY: BLINK INFORMATION / INFORMATION CLIGNOTEMENT LENT
   DFCCOM1 : BOOL ;	//FACILITY: COMMUNICATION CARD FAULT (CP340) / DEFAUT CARTE DE COMMUNICATION ETH
   DF_ILOT : BOOL ;	//FACILITY: FAULT / DEFAUT ILOT
  END_STRUCT ;	
BEGIN
// 50 bytes; values not shown
END_DATA_BLOCK

ORGANIZATION_BLOCK OB 1
TITLE = "Main Program Sweep (Cycle)"
VERSION : 0.1
VAR_TEMP
  OB1_EV_CLASS : BYTE ;	//Bits 0-3 = 1 (Coming event), Bits 4-7 = 1 (Event class 1)
  OB1_SCAN_1 : BYTE ;	//1 (Cold restart scan 1 of OB 1), 3 (Scan 2-n of OB 1)
  OB1_PRIORITY : BYTE ;	//Priority of OB Execution
  OB1_OB_NUMBR : BYTE ;	//1 (Organization block 1, OB1)
  OB1_RESERVED_1 : BYTE ;	//Reserved for system
  OB1_RESERVED_2 : BYTE ;	//Reserved for system
  OB1_PREV_CYCLE : INT ;	//Cycle time of previous OB1 scan (milliseconds)
  OB1_MIN_CYCLE : INT ;	//Minimum cycle time of OB1 (milliseconds)
  OB1_MAX_CYCLE : INT ;	//Maximum cycle time of OB1 (milliseconds)
  OB1_DATE_TIME : DATE_AND_TIME ;	//Date and time OB1 started
END_VAR
BEGIN
// (block stored without names or comments; labels and parameter names are numbered)
END_ORGANIZATION_BLOCK

SYMBOL_TABLE
"PRMPPB02"	C 1	COUNTER	// Pulsos para Reset MPP.MP.B02
"PRMPPB01"	C 2	COUNTER	// Pulsos para Reset MPP.MP.B01
"PRMPPA01"	C 3	COUNTER	// Pulsos para Reset MPP.MP.A01
"I01"	DB 1	FB 1	// FACILITY: INSTANCE DB (FB1)
"I02"	DB 2	FB 2	// FACILITY: INSTANCE DB FOR MMC CONTROL (FB2)
"I03"	DB 3	FB 3	// FACILITY: INSTANCE DB FOR MOP/LOP
"I04"	DB 4	FB 4	// FACILITY: INSTANCE DB FOR COMMUNICATION / DB D'INSTANCE POUR LA COMMUNICATION
"CDIV"	DB 69	DB 69	// FACILITY: DIVERSITIES CODES TABLE / TABLE CODES DIVERSITES
"SFM_DB"	DB 75	FB 20	// FACILITY: DB FAILURE MESSAGE (SFM_FB) LINK WITH PROFINET CONTROL
"SFM_GLOBAL_DB"	DB 76	DB 76	// DIAGNOSTIC BLOCK FOR THE SIGNALISATION OF THE SYSTEM ERRORS
"SFM_PN"	DB 77	DB 77	// PROFINET DIAGNOSTIC FUNCTION EDITING DB FOR IHMP
"SIP1"	DB 89	DB 89	// SIPTOL EXCHANGES DATAS / TABLE D'ECHANGES SIPTOL
"PILE"	DB 90	DB 90	// FACILITY: FIFO STORAGE / PILE DE STOCKAGE
"IDENT"	DB 93	DB 93	// RFID DATAS / IDENTIFIANT DYNAMIQUE
"IBD"	DB 95	DB 95	// FACILITY: DATA BASE DB / DB BASE DE DONNEE
"IIT"	DB 96	DB 96	// FACILITY: PART TABLE / DB TABLE PIECE
"IIS"	DB 97	DB 97	// FACILITY: SUPPORT WORD TABLE / DB MOTS SUPPORT
"IG"	DB 99	DB 99	// FACILITY: GLOBAL DB / DB GLOBAL
"Z1"	DB 100	FB 100	// ZONA 1: INSTANCE DB
"Z1A0L"	DB 109	FB 109	// A0 LANZAMIENTO BLOQUEO DE DATOS INSTANCIA
"Z1A01"	DB 110	FB 110	// A01 MONTAJE BLOQUEO DE DATOS INSTANCIA / BLOC DE DONNEES INSTANCE A01 MONTAJE
"Z1A11"	DB 111	FB 111	// A11 OP_BIMA BLOQUEO DE DATOS INSTANCIA / BLOC DE DONNEES INSTANCE A11 OP_BIMA
"Z1A12"	DB 112	FB 112	// A12 OP_BIMA BLOQUEO DE DATOS INSTANCIA / BLOC DE DONNEES INSTANCE A121 OP_BIMA
"Z1B0L"	DB 119	FB 119	// B0 LANZAMIENTO BLOQUEO DE DATOS INSTANCIA
"Z1B01"	DB 120	FB 120	// B01 MONTAJE BLOQUEO DE DATOS INSTANCIA / BLOC DE DONNEES INSTANCE B01 MONTAJE
"Z1B11"	DB 121	FB 121	// B11 OP_BIMA BLOQUEO DE DATOS INSTANCIA / BLOC DE DONNEES INSTANCE B11 OP_BIMA
"Z1B12"	DB 122	FB 122	// B12 OP_BIMA BLOQUEO DE DATOS INSTANCIA / BLOC DE DONNEES INSTANCE B12 OP_BIMA
"Z1B13"	DB 123	FB 123	// B13 OP_BIMA BLOQUEO DE DATOS INSTANCIA / BLOC DE DONNEES INSTANCE B13 OP_BIMA
"Z1C0R"	DB 129	FB 129	// C0 RECALAGE BLOQUEO DE DATOS INSTANCIA / BLOC DE DONNEES INSTANCE C0 RECALAGE
"Z1C01"	DB 130	FB 130	// C01 MONTAJE BLOQUEO DE DATOS INSTANCIA / BLOC DE DONNEES INSTANCE C01 MONTAJE
"Z1C11"	DB 131	FB 131	// C11 OP_BIMA BLOQUEO DE DATOS INSTANCIA / BLOC DE DONNEES INSTANCE C11 OP_BIMA
"Z1C12"	DB 132	FB 132	// C12 OP_BIMA BLOQUEO DE DATOS INSTANCIA / BLOC DE DONNEES INSTANCE C12 OP_BIMA
"Z1C13"	DB 133	FB 133	// C13 OP_BIMA BLOQUEO DE DATOS INSTANCIA / BLOC DE DONNEES INSTANCE C13 OP_BIMA
"Z1C0V"	DB 134	FB 134
"Z1C0M"	DB 135	FB 135
"Z1B02"	DB 140	FB 140	// B02 MONTAJE BLOQUEO DE DATOS INSTANCIA / BLOC DE DONNEES INSTANCE B02 MONTAJE
"Z1B21"	DB 141	FB 141	// B21 OP_BIMA BLOQUEO DE DATOS INSTANCIA / BLOC DE DONNEES INSTANCE B21 OP_BIMA
"Z1B22"	DB 142	FB 142	// B22 OP_BIMA BLOQUEO DE DATOS INSTANCIA / BLOC DE DONNEES INSTANCE B22 OP_BIMA
"Z1B23"	DB 143	FB 143	// B23 OP_BIMA BLOQUEO DE DATOS INSTANCIA / BLOC DE DONNEES INSTANCE B23 OP_BIMA
"Z1C02"	DB 150	FB 150	// C02 MONTAJE BLOQUEO DE DATOS INSTANCIA / BLOC DE DONNEES INSTANCE C02 MONTAJE
"Z1C21"	DB 151	FB 151	// C21 OP_BIMA BLOQUEO DE DATOS INSTANCIA / BLOC DE DONNEES INSTANCE C21 OP_BIMA
"Z1C22"	DB 152	FB 152	// C22 OP_BIMA BLOQUEO DE DATOS INSTANCIA / BLOC DE DONNEES INSTANCE C22 OP_BIMA
"Z1C23"	DB 153	FB 153	// C23 OP_BIMA BLOQUEO DE DATOS INSTANCIA / BLOC DE DONNEES INSTANCE C23 OP_BIMA
"Z1T"	DB 198	DB 198	// ZONA 1: REFERENCE TIME FOR MOVEMENTS
"Z1G"	DB 199	DB 199	// ZONA 1: GLOBAL DB
"A01LwTALO"	DB 950	DB 950	// Amw LOCAL TABLE / TABLE LOCALE
"A01TALO"	DB 951	DB 951	// A01: LOCAL TABLE / TABLE LOCALE
"A01wTALO"	DB 952	DB 952	// A01w: LOCAL TABLE / TABLE LOCALE
"B01TALO"	DB 953	DB 953	// B01: LOCAL TABLE / TABLE LOCALE
"B01wTALO"	DB 954	DB 954	// B01w: LOCAL TABLE / TABLE LOCALE
"C01TALO"	DB 955	DB 955	// C01: LOCAL TABLE / TABLE LOCALE
"C01wTALO"	DB 956	DB 956	// C01w: LOCAL TABLE / TABLE LOCALE
"B02TALO"	DB 957	DB 957	// B02: LOCAL TABLE / TABLE LOCALE
"B02wTALO"	DB 958	DB 958	// B02w: LOCAL TABLE / TABLE LOCALE
"C02TALO"	DB 959	DB 959	// C02: LOCAL TABLE / TABLE LOCALE
"C02wTALO"	DB 960	DB 960	// C02w: LOCAL TABLE / TABLE LOCALE
"D01TALO"	DB 961	DB 961	// D01: LOCAL TABLE / TABLE LOCALE
"D01wTALO"	DB 962	DB 962	// D01w: LOCAL TABLE / TABLE LOCALE
"ITR0"	DB 1000	FB 1000	// FACILITY: INSTANCE DB FOR SAFETY OPERATOR CONTROL (FB1000)
"ITRZ1SOP"	DB 1010	FB 1010	// Z1: INSTANCE DB FOR SAFETY OPERATOR CONTROL / DB D'INSTANCE SECU OP
"ITRZ1SOPTR"	DB 1011	FB 1011	// ZONA 1 : DB Instance Gestion SAFETY Sécurité opérateur (RSOP) de la ZONA 1
"TRM"	DB 1098	DB 1098	// FACILITY: SAFETY OPERATOR CONTROL
"TRI"	DB 1099	DB 1099	// FACILITY: SAFETY OPERATOR PROCESSING DB
"ITS0"	DB 1100	FB 1100	// FACLITY: SAFETY CONTROL DB
"ITSZ1_AU_ES_FZ"	DB 1110	FB 1110	// ZONA 1: SAFETY CONTROL INSTANCE DB EMERGENCY STOP (AU)
"ITSZ1_SOP"	DB 1111	FB 1111	// ZONA 1: SAFETY CONTROL INSTANCE DB STARTING-UP (ES)
"TSM"	DB 1279	DB 1279	// FACILITY: SAFETY CONTROL DB
"TSE_AVAL"	DB 1288	FB 1692	// STD - INSTANCIA DB OF FB 1692 (F_SENDDP) SAFETY DATA SEND
"TSR_AVAL"	DB 1289	FB 1693	// STD - INSTANCIA DB OF FB 1693 (F_RCVDP) SAFETY DATA RECEIVE
"TNI"	DB 1290	DB 1290	// STD.EXCHANGE DB BETWEEN SAFETY GROUPS OB 32 -> OB 34
"TNZ1"	DB 1291	DB 1291
"F_GLOBDB"	DB 1300	DB 1300	// F_: F_Global_Data Block
"F00250__B01SB___M11"	DB 1301	FB 1300
"F00244__B01SB___M10"	DB 1302	FB 1300
"F00238__B01SB___M09"	DB 1303	FB 1300
"F00232__B01SB___M08"	DB 1304	FB 1300
"F00108__Z1ZB___M07"	DB 1305	FB 1300
"F00102__Z1ZB___M06"	DB 1306	FB 1300
"F00214__A01SB___M10"	DB 1308	FB 1300
"F00208__A01SB___M09"	DB 1309	FB 1300
"F00202__A01SB___M08"	DB 1310	FB 1300
"F00220__A01SB___M11"	DB 1311	FB 1300
"F00310__B02SB___M11"	DB 1312	FB 1300
"F00304__B02SB___M10"	DB 1313	FB 1300
"F00298__B02SB___M09"	DB 1314	FB 1300
"F00292__B02SB___M08"	DB 1315	FB 1300
"F00262__C01SB___M08"	DB 1316	FB 1300
"F00268__C01SB___M09"	DB 1317	FB 1300
"F00274__C01SB___M10"	DB 1318	FB 1300
"F00280__C01SB___M11"	DB 1319	FB 1300
"F00322__C02SB___M08"	DB 1320	FB 1300
"F00328__C02SB___M09"	DB 1321	FB 1300
"F00334__C02SB___M10"	DB 1322	FB 1300
"F00340__C02SB___M11"	DB 1323	FB 1300
"Z1MPDEV"	DB 1600	DB 1600	// PALABRA PIEZA ESPECIFICA MARCHA VACIO
"AFF"	DB 1863	DB 1863	// SIEBERT DISPLAY STRING STORAGE / ALMACENAMIENTO MENSAJE VISULIZADOR SIEBERT
"DB_IHM_WINCC"	DB 1962	FB 1962	// FACILITY: HMI INTERFACING WINCCFLEXIBLE RT
"DB_MMC"	DB 2000	DB 2000	// BACKUP COPY AND RESTORE OF EXTERN MEMORY MAP (MMC)
"DB_MMCZ1T"	DB 2001	DB 2001	// Sauvegarde et restitution sur carte mémoire (MMC) des temps d'apprentissage Z1
"TALO"	DB 2005	DB 2005	// LOCAL TABLE
"DB_OPMAINT"	DB 2022	FB 2022	// MAINTENANCE SCREEN CONTROL MOP ou LOP PANEL
"DB_PN"	DB 2036	FB 2036	// INSTANCE IO PROFINET DB
"0_01_ILOT"	FB 1	FB 1	// FACILITY: FACILITY MANAGEMENT
"0_02_MMC"	FB 2	FB 2	// FACILITY: BACKUP MANAGEMENT AND DATA RESTITUTION ON EXTERNAL MMC CARD
"0_03_XOP"	FB 3	FB 3	// FACILITY: MOP/LOP MANAGEMENT
"0_04_COM"	FB 4	FB 4	// FACILITY: COM CONTROL WITH SIPTOL / GESTION DE LA COMMUNICATION AVEC SIPTOL
"SFM_FB"	FB 20	FB 20	// DIAGNOSTIC BLOCK FOR SYSTEM ERRORS SIGNALLING
"1_00_ZONA1"	FB 100	FB 100	// ZONA 1: ZONA CONTROL
"1_A0_LANZAMIENTO"	FB 109	FB 109	// A0 LANZAMIENTO FUNCTION BLOC / SECTION PROGRAMME A0 LANZAMIENTO
"1_A01_MONTAJE"	FB 110	FB 110	// A01 MONTAJE FUNCTION BLOC / SECTION PROGRAMME A01 MONTAJE
"1_A11_OP"	FB 111	FB 111	// A01 OP_A11 FUNCTION BLOC / SECTION PROGRAMME A01 OP_A11
"1_A12_OP"	FB 112	FB 112	// A01 OP_A12 FUNCTION BLOC / SECTION PROGRAMME A01 OP_A12
"1_B0_LANZAMIENTO"	FB 119	FB 119	// B0 LANZAMIENTO FUNCTION BLOC / SECTION PROGRAMME B0 LANZAMIENTO
"1_B01_MONTAJE"	FB 120	FB 120	// B01 MONTAJE FUNCTION BLOC / SECTION PROGRAMME B01 MONTAJE
"1_B11_OP"	FB 121	FB 121	// B01 OP_B11 FUNCTION BLOC / SECTION PROGRAMME B01 OP_B11
"1_B12_OP"	FB 122	FB 122	// B01 OP_B12 FUNCTION BLOC / SECTION PROGRAMME B01 OP_B12
"1_B13_OP"	FB 123	FB 123	// B01 OP_B13 FUNCTION BLOC / SECTION PROGRAMME B01 OP_B13
"1_C0_RECALAGE"	FB 129	FB 129	// C0 RECALAGE FUNCTION BLOC / SECTION PROGRAMME C0 RECALAGE
"1_C01_MONTAJE"	FB 130	FB 130	// C01 MONTAJE FUNCTION BLOC / SECTION PROGRAMME C01 MONTAJE
"1_C11_OP"	FB 131	FB 131	// C01 OP_C11 FUNCTION BLOC / SECTION PROGRAMME C01 OP_C11
"1_C12_OP"	FB 132	FB 132	// C01 OP_C12 FUNCTION BLOC / SECTION PROGRAMME C01 OP_C12
"1_C13_OP"	FB 133	FB 133	// C01 OP_C13 FUNCTION BLOC / SECTION PROGRAMME C01 OP_C13
"1_C0_VISU"	FB 134	FB 134
"1_C0_MARIAGE"	FB 135	FB 135
"1_B02_MONTAJE"	FB 140	FB 140	// B02 MONTAJE FUNCTION BLOC / SECTION PROGRAMME B02 MONTAJE
"1_B21_OP"	FB 141	FB 141	// B02 OP_B21 FUNCTION BLOC / SECTION PROGRAMME B02 OP_B21
"1_B22_OP"	FB 142	FB 142	// B02 OP_B22 FUNCTION BLOC / SECTION PROGRAMME B02 OP_B22
"1_B23_OP"	FB 143	FB 143	// B02 OP_B23 FUNCTION BLOC / SECTION PROGRAMME B02 OP_B23
"1_C02_MONTAJE"	FB 150	FB 150	// C02 MONTAJE FUNCTION BLOC / SECTION PROGRAMME C02 MONTAJE
"1_C21_OP"	FB 151	FB 151	// C02 OP_C21 FUNCTION BLOC / SECTION PROGRAMME C02 OP_C21
"1_C22_OP"	FB 152	FB 152	// C02 OP_C22 FUNCTION BLOC / SECTION PROGRAMME C02 OP_C22
"1_C23_OP"	FB 153	FB 153	// C02 OP_C23 FUNCTION BLOC / SECTION PROGRAMME C02 OP_C23
"F_TON"	FB 185	FB 185	// F_: Timer Switch On Delay
"F_TOF"	FB 186	FB 186	// F_: Timer Switch Of Delay
"TR0"	FB 1000	FB 1000	// FACILITY: SAFETY OPERATOR CONTROL FB
"TRZ1SOP"	FB 1010	FB 1010	// Z1: INSTANCE FB FOR SAFETY OPERATOR CONTROL / FB D'INSTANCE SECU OP
"TS0"	FB 1100	FB 1100	// FACILITY: SAFETY CONTROL FB
"TSZ1_AU_ES_FZ"	FB 1110	FB 1110	// ZONA 1: SAFETY CONTROL INSTANCE DB EMERGENCY STOP (AU)
"TSZ1_SOP"	FB 1111	FB 1111	// ZONA 1: SAFETY CONTROL INSTANCE DB STARTING-UP (ES)
"F_IO_CGP"	FB 1300	FB 1300	// F_: Driver Block In-Output with CANAL Granular Passivation
"F_CTRL_1"	FB 1301	FB 1301	// F_: Test Block an Programm Run Control 1
"F_CTRL_2"	FB 1302	FB 1302	// F_: Test Block an Programm Run Control 2
"FITON"	FB 1303	FB 1303
"FI2HAND"	FB 1304	FB 1304
"FIACK_GL"	FB 1305	FB 1305
"F_DIAG_N"	FB 1307	FB 1307	// F_: Diagnosticbuffer Message with non CPU-Stop
"BFI_DEVERM"	FB 1600	FB 1600	// Gestion du déverminage d'une table
"TUSEND"	FB 1681	FB 1681	// Send Data via UDP
"TCON"	FB 1685	FB 1685	// Connect
"F_2HAND"	FB 1688	FB 1688
"F_SENDDP"	FB 1692	FB 1692
"F_RCVDP"	FB 1693	FB 1693
"F_ACK_GL"	FB 1695	FB 1695	// ACKNOWLEDGE OF ALL PERIPHERALS F / ACQUITTEMENT GLOBAL PERIPH F
"P_SEND"	FB 1698	FB 1698	// SEND DATA TO CP340 / ENVOI DE DONNEES VERS LES CARTES CP 340 - LEAN
"P_RCV"	FB 1699	FB 1699	// RECEIVE DATA FROM CP340 / RECEPTION DE DONNEES DEPUIS LES CARTES CP 340 - LEAN
"BFS_BSEC"	FB 1700	FB 1700	// BFS - Zx : Traitement SAFETY des relais de sécurité (RAU, RMS, RFZ, RL)
"BFS_BSECTR"	FB 1701	FB 1701	// DELAYED SAFETY RELAY PROCESSING (RMSTR) / TRAITEMENT RELAIS SECU TEMPORISE
"BFS_PORTE"	FB 1702	FB 1702	// BFS - ZX: ACCESS DOOR SAFETY PROCESSING / TRAITEMENT SAFETY PORTILLON D'ACCES
"BFS_CR"	FB 1705	FB 1705	// BFS - FEEDBACK CONTROL (F-RO) / CONTROLE RETOUR (F-RO)
"BFS_MUT"	FB 1707	FB 1707
"BFS_BSEC1"	FB 1710	FB 1710
"BFS_BSECTR1"	FB 1711	FB 1711
"BFS_PUERTA1"	FB 1712	FB 1712
"BFS_AIR1"	FB 1713	FB 1713
"BFS_CRM1"	FB 1714	FB 1714
"BFS_CR1"	FB 1715	FB 1715
"BFS_LEVA_ROBOT1"	FB 1716	FB 1716
"BFS_ROB_KUKA_PS"	FB 1720	FB 1720
"BFS_Minomi"	FB 1750	FB 1750	// Gestión de la seguridad de un carro Minomi (Despaletización)
"BF_DEVERM"	FB 1803	FB 1803	// BF STAGE DRY RUN CONTROL / BF GESTION DEVERMINAGE POSTE
"BF_PNPN_MESG"	FB 1852	FB 1852	// SEND RECEIVE MESSAGE BY PNPN INTERFACE/ EMISION RECEPCION MENSAJE VIA PNPN
"BF_G120DS_V2"	FB 1853	FB 1853	// G120D DRIVE BOX CONTROL / GESTION COFRE VAR G120D
"BF_G120S_V2"	FB 1854	FB 1854	// G120 DRIVE PLATE CONTROL / GESTION PLETINA VAR G120
"BF_CARACT_SIEBERT"	FB 1856	FB 1856	// SIEBERT DISPLAY MESSAGE CONFIGURATION / MISE EN FORME MESSAGE AFFICHEUR SIEBERT
"BF_RECALAGE2"	FB 1857	FB 1857	// Gestion des points de recalage
"BF_LANZAMIENTO"	FB 1858	FB 1858	// GESTION LANZAMIENTO SIPTOL
"BF_AFF SIEBERT (2*13) PN"	FB 1860	FB 1860	// VISUALIZADOR 2 LINEAS DE 13 CARACTERES
"BF_DP_LOCATOR"	FB 1866	FB 1866	// DP_LOCATOR CONTROL / GESTION DES DP_LOCATOR
"BF_WELDING_BOX"	FB 1868	FB 1868	// WELDING BOX CONTROL / GESTION DE COFRES PARAMETROS SOLDADURA
"BF_CONF_MACHINE"	FB 1869	FB 1869	// GESTION BASE DE DATOS CONFIGURACION MAQUINA
"BF_CODE_PROCESS"	FB 1870	FB 1870	// GESTION BASE DE DONNEE CODE PROCESS
"BF_DATABASE3"	FB 1871	FB 1871	// DATABASE MANAGEMENT / GESTION BASE DE DONNEES
"BF_IHMMUT1"	FB 1874	FB 1874	// Diagnostico IHM(P) BFS_MUT1
"BF_IHMLEVA_ROBOT1"	FB 1875	FB 1875	// BF control buen FUNCIONAMIENTO de la LEVA robot
"BF_IHMCR1"	FB 1876	FB 1876	// BF control IHM del RELE no pilotado por el API pero controlado
"BF_IHMCRM1"	FB 1877	FB 1877	// BF control IHM del RELE de control union de masa CRM
"BF_S120_S"	FB 1892	FB 1892
"BF_CABRS"	FB 1897	FB 1897	// BARCODIGO READER / LECTOR DE CODIGO DE BARRAS
"BF_IHMPUERTA1"	FB 1930	FB 1930	// BF - ZONA : Diagnóstico del bloque BFS_IHMPUERTA
"BF_IHMAIR1"	FB 1931	FB 1931	// BF - ZONA : Diagnóstico del bloque BFS_IHMAIR
"BF_ZONA_MODE_IHM1"	FB 1932	FB 1932	// ZONA: Tratamiento de modos y de pupitres de cde manu de la  ZONA
"BF_MOUV_PL2M"	FB 1937	FB 1937	// Mesa giratoria - 2 Montajes / 2 Sentidos
"BF_IHMCRM"	FB 1942	FB 1942	// BF gérant l'IHM du relais de controçle raccordement de masse CRM
"BF_IHMBSEC"	FB 1944	FB 1944	// BF - ZONA : Diagnostic SAFETY BFS_BSEC
"BF_IHMAIR"	FB 1948	FB 1948	// BF - ZONA : Diagnostic du bloc BFS_IHMAIR
"BF_RB_COD_PREH_API"	FB 1953	FB 1953	// Gestion de garra por API (secuencias 1 a 16)
"BF_MODBUS MASTER CP340"	FB 1958	FB 1958	// Modbus Maitre sur CP 340 (liaison serie)
"BF_MODBUS SLAVE CP340"	FB 1959	FB 1959	// Modbus Esclave avec CP 340
"BF_Modbus_TCP_Master"	FB 1960	FB 1960	// BF gerant le protocole MODBUS TCP/IP en tant que Client TCP et Maitre MODBUS
"BF_MODBUS TCPIP SLAVE"	FB 1961	FB 1961	// Esclave Modbus sur CP Ethernet
"BF_IHM_WINCC"	FB 1962	FB 1962	// BF- GESTION IMAGENES WINCC FLEXIBLE
"BF_ZONA_MODE_IHM"	FB 1963	FB 1963	// ZONA: Traitement des Modes et des pupitre de cde manu de la  ZONA
"BF_RB_SERVICIO"	FB 1997	FB 1997	// BF- Envio de un GRUPO de robot a fresado
"BF_MMC"	FB 2000	FB 2000	// SALVAGUARDA Y RESTITUCION MEMORIA SOBRE CARTA MEMORIA EXTERNA (MMC)
"BF_MB_CADENA1"	FB 2001	FB 2001	// PILOTAJE DEL MOTOR DEL MUEBLE Y VIGILANCIA DE DEFECTOS
"BF_MB_TOPE1"	FB 2002	FB 2002	// MUEBLE ACUMULACION - PILOTAJE DE UN TOPE
"BF_MARIAGE_API"	FB 2003	FB 2003	// Gestion des Mariados Pieza
"BF_ILOT"	FB 2004	FB 2004	// BF- Gestion info lié à l'installation ( Ilot )
"BF_DATABASE1"	FB 2005	FB 2005	// Gestionde Base de Données
"BF_B_VIEAPI"	FB 2006	FB 2006	// CONTROL DE LA COMUNICACION ENTRE DOS AUTOMATAS ENLAZADOS
"BF_TOPE_CONVOYEUR2"	FB 2007	FB 2007	// PILOTAJE DE UN TOPE
"BF_IDENT"	FB 2015	FB 2015	// LECTURA/ESCRITURA DE ETIQUETAS RFID
"BF_ROBOT"	FB 2016	FB 2016	// Interface API <=> Robot Version 1.2a
"BF_TCY_SUIV"	FB 2019	FB 2019	// MEDIDA LES TIEMPO DE CICLO DE UN MEDIO DE PRODUCCION
"BF_RUP_FLU"	FB 2020	FB 2020	// SEGUIMIENTO-RUPTURA DE FLUJO
"BF_CPT_PIECE"	FB 2021	FB 2021	// BF- Compteur de pièce
"BF_OPMAINT"	FB 2022	FB 2022	// gestion écrans maintenance pupitre MOP ou LOP
"BF_API_MAITRE_CAL"	FB 2031	FB 2031	// Gestion del Diálogo API MAESTRO CAL
"BF_ACT_DESACT"	FB 2033	FB 2033	// BF- ACTIVACION DESACTIVACION DE UN IO DISPOSITIVO
"BF_DIAG_PROFINET"	FB 2036	FB 2036	// BF- DIAGNOSTICO PROFINET IO
"BF_TF_TP"	FB 2037	FB 2037	// TRANSFERENCIA DE TABLA DE MEMORIAS PIEZAS
"BF_FIFO"	FB 2039	FB 2039	// ASEGURA LA GESTION DE UNA PILA FIFO
"BF_MVSE2P1"	FB 2040	FB 2040	// GESTION DE UN MOVIMIENTO SIMPLE EFECTO 2 POSICIONES
"BF_MOUVMP1"	FB 2041	FB 2041	// GESTION DE UN MOVIMIENTO MULTI POSICION
"BF_MOUV2P1"	FB 2042	FB 2042	// BF- GESTION DE UN MOVIMIENTO A 2 POSICIONES
"0_00_CYCLO_ISLA"	FC 1	FC 1	// FACILITY: CALL OF FACILITY FB
"0_11_SECU_FERMEE"	FC 11	FC 11	// COPY OF SAFETY INFORMATION ZONA 1 TO 9 FOR THE SAFETY CLOSED ZONA
"SFM_FC"	FC 22	FC 22	// BLOCK DIAGNOSTIC FOR ERROR REPORTING SYSTEM
"1_00_CYCLO_Z1"	FC 100	FC 100	// ZONA 1: CALL OF FB ZONA
"0_00_TRSAFETY"	FC 1000	FC 1000	// STD - FACILITY: EXECUTION F GROUP ASSOCIATE TO OB34 (FAST TASK)
"0_00_TRCYCLE"	FC 1001	FC 1001	// CALL OPERATOR ZONA FB LINKED IN FACILITY
"0_00_TSSAFETY"	FC 1100	FC 1100	// STD - FACILITY: EXECUTION F GROUP ASSOCIATE TO OB32 (NORMAL TASK)
"0_00_TSCICLO"	FC 1101	FC 1101	// CALL OPERATOR NOT IN ZONA FB LINKED IN FACILITY
"AG_SEND"	FC 1698	FC 1698	// AG SEND
"AG_RECV"	FC 1699	FC 1699	// AG RECEIVE
"BADI"	I 0.0	BOOL	// (MOP-IM.M01-02): PULSADOR ANULACION DEFECTO
"BRI"	I 0.1	BOOL	// (MOP-IM.M01-02): PULSADOR REARME ISLA
"Z1BMCY"	I 0.2	BOOL	// (MOP-IM.M01-02): PULSADOR MARCHA CICLO
"Z1SMM"	I 0.3	BOOL	// (MOP-IM.M01-02): SELECTOR MODO MANUAL
"Z1SMA"	I 1.0	BOOL	// (MOP-IM.M01-02): SELECTOR MODO AUTO
"Z1BMR1"	I 1.1	BOOL	// (MOP-IM.M01-02): PULSADOR RETROCESO MOVIMIENTO
"Z1BMA1"	I 1.2	BOOL	// (MOP-IM.M01-02): PULSADOR AVANCE MOVIMIENTO
"CLIMOK"	I 1.3	BOOL	// (Z1MOP): AIRE CONDITIONAR
"Z1CCFRO1"	I 100.0	BOOL	// (Z1ZB.M02):  (Z1F-R01) CONTROL COMUN AU
"Z1CCFRO2"	I 100.1	BOOL	// (Z1ZB.M02):  (Z1F-R02) CONTROL COMUN ES
"Z1CCB24Z"	I 100.2	BOOL	// (Z1ZB.M02): RETORNO CONTROL DISYUNTOR 24V (24Z)
"Z1CCB24R"	I 100.3	BOOL	// (Z1ZB.M02): RETORNO CONTROL DISYUNTOR 24V (24R)
"C0RVALOP1"	I 100.6	BOOL	// (Z1ZB.M02): PULSADOR VALIDACCION OPERADOR POR EL RECALAGE
"C0RVALOP2"	I 100.7	BOOL	// (Z1ZB.M02): PULSADOR CONFIRMACION OPERADOR POR EL RECALAGE
"Z1CP7B"	I 101.0	BOOL	// (Z1ZB.M03): CONTROL PRESION 7 BARS
"Z1CRM"	I 101.1	BOOL	// (Z1ZB.M03): CONTROL RELE DE MASA
"BAUI"	I 102.0	BOOL	// (Z1ZB.M06): PULSADOR PARADA DE EMERGENCIA MOP
"Z1SSZ"	I 102.2	BOOL	// (Z1ZB.M06): SELECTOR DE SEGURIDAD
"Z1IFRO1"	I 113.0	BOOL	// (Z1ZB.M08): F-RO1 INTERNAL CONTROL
"Z1IFRO2"	I 114.0	BOOL	// (Z1ZB.M09): F-RO2 INTERNAL CONTROL
"A01CCFRO1"	I 200.0	BOOL	// (A01SB.M02): CONTROL COMUN SOP
"A01CCFRO2"	I 200.1	BOOL	// (A01SB.M02): SAFETY COMMON CONTROL 2
"A01CCFRO3"	I 200.2	BOOL	// (A01SB.M02): SAFETY COMMON CONTROL 3
"A0DCZA"	I 200.3	BOOL	// info guinche en zona A
"A01CCB24Z"	I 200.4	BOOL	// (A01SB.M02): RETORNO CONTROL DISYUNTOR 24V (24Z)
"A01CCB24R"	I 200.5	BOOL	// (A01SB.M02): RETORNO CONTROL DISYUNTOR 24V (24R)
"A0DCZB"	I 200.6	BOOL	// info guinche en zona B
"A0DCZC"	I 200.7	BOOL	// info guinche en zona C
"A01BROC"	I 201.4	BOOL	// (A01SB.M03): PULSADOR DEMANDA RETORNO ORIGEN DE CICLO
"A0CCVL52"	I 201.5	BOOL	// CILINDRO CAMBIO DE VIA POS L52
"A0CCVB52"	I 201.6	BOOL	// CILINDRO CAMBIO DE VIA POS B52
"A11BAU1"	I 202.0	BOOL	// (A01SB.M08): PULSADOR  PARADA EMERGENCIA OPERARIO A11
"A12BAU1"	I 202.1	BOOL	// (A01SB.M08): PULSADOR  PARADA EMERGENCIA OPERARIO A12
"A11BP11"	I 208.0	BOOL	// (A01SB.M09): PULSADOR 1 DE VALIDACION OPERARIO 1 (CANAL1)
"A11BP21"	I 208.1	BOOL	// (A01SB.M09): PULSADOR 2 DE VALIDACION OPERARIO  1 (CANAL1)
"A12BP11"	I 208.2	BOOL	// (A01SB.M09): PULSADOR 1 DE VALIDACION OPERARIO 2 (CANAL 1)
"A12BP21"	I 208.3	BOOL	// (A01SB.M09): PULSADOR 2 DE VALIDACION OPERARIO 2 (CANAL 1)
"A11BP12"	I 208.4	BOOL	// (A01SB.M09): PULSADOR 1 DE VALIDACION OPERARIO 1 (CANAL2)
"A11BP22"	I 208.5	BOOL	// (A01SB.M09): PULSADOR 2 DE VALIDACION OPERARIO  1 (CANAL2)
"A12BP12"	I 208.6	BOOL	// (A01SB.M09): PULSADOR 1 DE VALIDACION OPERARIO 2 (CANAL 2)
"A12BP22"	I 208.7	BOOL	// (A01SB.M09): PULSADOR 2 DE VALIDACION OPERARIO 2 (CANAL 2)
"A01IFRO1"	I 225.0	BOOL	// (A01SB.M12): CONTROL COMUN SOP
"A01IFRO2"	I 226.0	BOOL	// (A01SB.M12): CONTROL COMUN 2
"A01IFRO3"	I 227.0	BOOL	// (A01SB.M12): CONTROL COMUN 3
"B01CCFRO1"	I 230.0	BOOL	// (B01SB.M02): CONTROL COMUN SOP
"B01CCFRO2"	I 230.1	BOOL	// (B01SB.M02): SAFETY COMMON CONTROL 2
"B01CCFRO3"	I 230.2	BOOL	// (B01SB.M02): SAFETY COMMON CONTROL 3
"B01CCB24Z"	I 230.4	BOOL	// (B01SB.M02): RETORNO CONTROL DISYUNTOR 24V (24Z)
"B01CCB24R"	I 230.5	BOOL	// (B01SB.M02): RETORNO CONTROL DISYUNTOR 24V (24R)
"B01BROC"	I 231.4	BOOL	// (B01SB.M03): PULSADOR DEMANDA RETORNO ORIGEN DE CICLO
"B11BAU1"	I 232.0	BOOL	// (B01SB.M08): PULSADOR  PARADA EMERGENCIA OPERARIO B11
"B12BAU1"	I 232.1	BOOL	// (B01SB.M08): PULSADOR  PARADA EMERGENCIA OPERARIO B12
"B13BAU1"	I 232.2	BOOL	// (B01SB.M08): PULSADOR  PARADA EMERGENCIA OPERARIO B13
"B11BP11"	I 238.0	BOOL	// (B01SB.M09): PULSADOR 1 DE VALIDACION OPERARIO 1 (CANAL1)
"B11BP21"	I 238.1	BOOL	// (B01SB.M09): PULSADOR 2 DE VALIDACION OPERARIO 1 (CANAL1)
"B12BP11"	I 238.2	BOOL	// (B01SB.M09): PULSADOR 1 DE VALIDACION OPERARIO 2 (CANAL1)
"B12BP21"	I 238.3	BOOL	// (B01SB.M09): PULSADOR 2 DE VALIDACION OPERARIO 2 (CANAL1)
"B11BP12"	I 238.4	BOOL	// (B01SB.M09): PULSADOR 1 DE VALIDACION OPERARIO 1 (CANAL2)
"B11BP22"	I 238.5	BOOL	// (B01SB.M09): PULSADOR 2 DE VALIDACION OPERARIO 1 (CANAL2)
"B12BP12"	I 238.6	BOOL	// (B01SB.M09): PULSADOR 1 DE VALIDACION OPERARIO 2 (CANAL2)
"B12BP22"	I 238.7	BOOL	// (B01SB.M09): PULSADOR 2 DE VALIDACION OPERARIO 2 (CANAL2)
"B13BP11"	I 244.0	BOOL	// (B01SB.M10): PULSADOR 1 DE VALIDACION OPERARIO 3 (CANAL1)
"B13BP21"	I 244.1	BOOL	// (B01SB.M10): PULSADOR 2 DE VALIDACION OPERARIO 3 (CANAL1)
"B13BP12"	I 244.4	BOOL	// (B01SB.M10): PULSADOR 1 DE VALIDACION OPERARIO 3 (CANAL2)
"B13BP22"	I 244.5	BOOL	// (B01SB.M10): PULSADOR 2 DE VALIDACION OPERARIO 3 (CANAL2)
"B01IFRO1"	I 255.0	BOOL	// (B01SB.M12): CONTROL COMUN SOP
"B01IFRO2"	I 256.0	BOOL	// (B01SB.M12): SAFETY COMMON 2
"B01IFRO3"	I 257.0	BOOL	// (B01SB.M12): SAFETY COMMON 3
"C01CCFRO1"	I 260.0	BOOL	// (C01SB.M02): CONTROL COMUN SOP
"C01CCFRO2"	I 260.1	BOOL	// (C01SB.M02): SAFETY COMMON CONTROL 2
"C01CCFRO3"	I 260.2	BOOL	// (C01SB.M02): SAFETY COMMON CONTROL 3
"C01CCB24Z"	I 260.4	BOOL	// (C01SB.M02): ELECTRICAL CIRCUIT BREAKER 24V (24Z)
"C01CCB24R"	I 260.5	BOOL	// (C01SB.M02): ELECTRICAL CIRCUIT BREAKER 24V (24R)
"C01DCRD"	I 260.6	BOOL	// (C01SB.M02): DETECTOR CRUZETA DESCARGA
"C01BROC"	I 261.4	BOOL	// (C01SB.M03): PULSADOR DEMANDA RETORNO ORIGEN DE CICLO
"C11BAU1"	I 262.0	BOOL	// (C01SB.M08): PULSADOR  PARADA EMERGENCIA OPERARIO C11
"C12BAU1"	I 262.1	BOOL	// (C01SB.M08): PULSADOR  PARADA EMERGENCIA OPERARIO C12
"C13BAU1"	I 262.2	BOOL	// (C01SB.M08): PULSADOR  PARADA EMERGENCIA OPERARIO C13
"C11BP11"	I 268.0	BOOL	// (C01SB.M09): PULSADOR 1 DE VALIDACION OPERARIO 1 (CANAL1)
"C11BP21"	I 268.1	BOOL	// (C01SB.M09): PULSADOR 2 DE VALIDACION OPERARIO 1 (CANAL1)
"C12BP11"	I 268.2	BOOL	// (C01SB.M09): PULSADOR 1 DE VALIDACION OPERARIO 2 (CANAL1)
"C12BP21"	I 268.3	BOOL	// (C01SB.M09): PULSADOR 2 DE VALIDACION OPERARIO 2 (CANAL1)
"C11BP12"	I 268.4	BOOL	// (C01SB.M09): PULSADOR 1 DE VALIDACION OPERARIO 1 (CANAL2)
"C11BP22"	I 268.5	BOOL	// (C01SB.M09): PULSADOR 2 DE VALIDACION OPERARIO 1 (CANAL2)
"C12BP12"	I 268.6	BOOL	// (C01SB.M09): PULSADOR 1 DE VALIDACION OPERARIO 2 (CANAL2)
"C12BP22"	I 268.7	BOOL	// (C01SB.M09): PULSADOR 2 DE VALIDACION OPERARIO 2 (CANAL2)
"C13BP11"	I 274.0	BOOL	// (C01SB.M10): PULSADOR 1 DE VALIDACION OPERARIO 3 (CANAL1)
"C13BP21"	I 274.1	BOOL	// (C01SB.M10): PULSADOR 2 DE VALIDACION OPERARIO 3 (CANAL1)
"C13BP12"	I 274.4	BOOL	// (C01SB.M10): PULSADOR 1 DE VALIDACION OPERARIO 3 (CANAL2)
"C13BP22"	I 274.5	BOOL	// (C01SB.M10): PULSADOR 2 DE VALIDACION OPERARIO 3 (CANAL2)
"C01IFRO1"	I 285.0	BOOL	// (C01SB.M12): CONTROL COMUN SOP
"C01IFRO2"	I 286.0	BOOL	// (C01SB.M12): SAFETY COMMON 2
"C01IFRO3"	I 287.0	BOOL	// (C01SB.M12): SAFETY COMMON 3
"B02CCFRO1"	I 290.0	BOOL	// (B02SB.M02): CONTROL COMUN SOP
"B02CCFRO2"	I 290.1	BOOL	// (B02SB.M02): SAFETY COMMON CONTROL 2
"B02CCFRO3"	I 290.2	BOOL	// (B02SB.M02): SAFETY COMMON CONTROL 3
"B02CCB24Z"	I 290.4	BOOL	// (B02SB.M02): ELECTRICAL CIRCUIT BREAKER 24V (24Z)
"B02CCB24R"	I 290.5	BOOL	// (B02SB.M02): ELECTRICAL CIRCUIT BREAKER 24V (24R)
"B02BROC"	I 291.4	BOOL	// (B02SB.M03): PULSADOR DEMANDA RETORNO ORIGEN DE CICLO
"B21BAU1"	I 292.0	BOOL	// (B02SB.M08): PULSADOR  PARADA EMERGENCIA OPERARIO C11
"B22BAU1"	I 292.1	BOOL	// (B02SB.M08): PULSADOR  PARADA EMERGENCIA OPERARIO C12
"B23BAU1"	I 292.2	BOOL	// (B02SB.M08): PULSADOR  PARADA EMERGENCIA OPERARIO C13
"B21BP11"	I 298.0	BOOL	// (B02SB.M09): PULSADOR 1 DE VALIDACION OPERARIO 1 (CANAL1)
"B21BP21"	I 298.1	BOOL	// (B02SB.M09): PULSADOR 2 DE VALIDACION OPERARIO 1 (CANAL1)
"B22BP11"	I 298.2	BOOL	// (B02SB.M09): PULSADOR 1 DE VALIDACION OPERARIO 2 (CANAL1)
"B22BP21"	I 298.3	BOOL	// (B02SB.M09): PULSADOR 2 DE VALIDACION OPERARIO 2 (CANAL1)
"B21BP12"	I 298.4	BOOL	// (B02SB.M09): PULSADOR 1 DE VALIDACION OPERARIO 1 (CANAL2)
"B21BP22"	I 298.5	BOOL	// (B02SB.M09): PULSADOR 2 DE VALIDACION OPERARIO 1 (CANAL2)
"B22BP12"	I 298.6	BOOL	// (B02SB.M09): PULSADOR 1 DE VALIDACION OPERARIO 2 (CANAL2)
"B22BP22"	I 298.7	BOOL	// (B02SB.M09): PULSADOR 2 DE VALIDACION OPERARIO 2 (CANAL2)
"B23BP11"	I 304.0	BOOL	// (B02SB.M10): PULSADOR 1 DE VALIDACION OPERARIO 3 (CANAL1)
"B23BP21"	I 304.1	BOOL	// (B02SB.M10): PULSADOR 2 DE VALIDACION OPERARIO 3 (CANAL1)
"B23BP12"	I 304.4	BOOL	// (B02SB.M10): PULSADOR 1 DE VALIDACION OPERARIO 3 (CANAL2)
"B23BP22"	I 304.5	BOOL	// (B02SB.M10): PULSADOR 2 DE VALIDACION OPERARIO 3 (CANAL2)
"B02IFRO1"	I 315.0	BOOL	// (B02SB.M12): CONTROL COMUN SOP
"B02IFRO2"	I 316.0	BOOL	// (B02SB.M12): SAFETY COMMON 2
"B02IFRO3"	I 317.0	BOOL	// (B02SB.M12): SAFETY COMMON 3
"C02CCFRO1"	I 320.0	BOOL	// (C02SB.M02): CONTROL COMUN SOP
"C02CCFRO2"	I 320.1	BOOL	// (C02SB.M02): SAFETY COMMON CONTROL 2
"C02CCFRO3"	I 320.2	BOOL	// (C02SB.M02): SAFETY COMMON CONTROL 3
"C02CCB24Z"	I 320.4	BOOL	// (C02SB.M02): ELECTRICAL CIRCUIT BREAKER 24V (24Z)
"C02CCB24R"	I 320.5	BOOL	// (C02SB.M02): ELECTRICAL CIRCUIT BREAKER 24V (24R)
"C02DCRD"	I 320.6	BOOL	// (C02SB.M02): DETECTOR CRUZETA DESCARGA
"C02BROC"	I 321.4	BOOL	// (C02SB.M03): PULSADOR DEMANDA RETORNO ORIGEN DE CICLO
"C21BAU1"	I 322.0	BOOL	// (C02SB.M08): PULSADOR  PARADA EMERGENCIA OPERARIO C11
"C22BAU1"	I 322.1	BOOL	// (C02SB.M08): PULSADOR  PARADA EMERGENCIA OPERARIO C12
"C23BAU1"	I 322.2	BOOL	// (C02SB.M08): PULSADOR  PARADA EMERGENCIA OPERARIO C13
"C21BP11"	I 328.0	BOOL	// (C02SB.M09): PULSADOR 1 DE VALIDACION OPERARIO 1 (CANAL1)
"C21BP21"	I 328.1	BOOL	// (C02SB.M09): PULSADOR 2 DE VALIDACION OPERARIO 1 (CANAL1)
"C22BP11"	I 328.2	BOOL	// (C02SB.M09): PULSADOR 1 DE VALIDACION OPERARIO 2 (CANAL1)
"C22BP21"	I 328.3	BOOL	// (C02SB.M09): PULSADOR 2 DE VALIDACION OPERARIO 2 (CANAL1)
"C21BP12"	I 328.4	BOOL	// (C02SB.M09): PULSADOR 1 DE VALIDACION OPERARIO 1 (CANAL2)
"C21BP22"	I 328.5	BOOL	// (C02SB.M09): PULSADOR 2 DE VALIDACION OPERARIO 1 (CANAL2)
"C22BP12"	I 328.6	BOOL	// (C02SB.M09): PULSADOR 1 DE VALIDACION OPERARIO 2 (CANAL2)
"C22BP22"	I 328.7	BOOL	// (C02SB.M09): PULSADOR 2 DE VALIDACION OPERARIO 2 (CANAL2)
"C23BP11"	I 334.0	BOOL	// (C02SB.M10): PULSADOR 1 DE VALIDACION OPERARIO 3 (CANAL1)
"C23BP21"	I 334.1	BOOL	// (C02SB.M10): PULSADOR 2 DE VALIDACION OPERARIO 3 (CANAL1)
"C23BP12"	I 334.4	BOOL	// (C02SB.M10): PULSADOR 1 DE VALIDACION OPERARIO 3 (CANAL2)
"C23BP22"	I 334.5	BOOL	// (C02SB.M10): PULSADOR 2 DE VALIDACION OPERARIO 3 (CANAL2)
"C02IFRO1"	I 345.0	BOOL	// (C02SB.M12): CONTROL COMUN SOP
"C02IFRO2"	I 346.0	BOOL	// (C02SB.M12): SAFETY COMMON 2
"C02IFRO3"	I 347.0	BOOL	// (C02SB.M12): SAFETY COMMON 3
"A01DEPLA1"	I 400.0	BOOL	// (A01E11) : DETECTOR RETROCESO PILOTO A1
"A01DDPLB1"	I 400.1	BOOL	// (A01E11) : DETECTOR RETROCESO PILOTO B1
"A01DDPLB2"	I 400.2	BOOL	// (A01E11) : DETECTOR RETROCESO PILOTO B2
"A01DDPLB3"	I 400.3	BOOL	// (A01E11) : DETECTOR RETROCESO PILOTO B3
"A01DDPLA1"	I 400.4	BOOL	// (A01E11) : DETECTOR AVANCE PILOTO A1
"A01DEPLB1"	I 400.5	BOOL	// (A01E11) : DETECTOR AVANCE PILOTO B1
"A01DEPLB2"	I 400.6	BOOL	// (A01E11) : DETECTOR AVANCE PILOTO B2
"A01DEPLB3"	I 400.7	BOOL	// (A01E11) : DETECTOR AVANCE PILOTO B3
"A01DDPLB4"	I 401.0	BOOL	// (A01E12) : DETECTOR RETROCESO PILOTO B4
"A01DDPLB5"	I 401.1	BOOL	// (A01E12) : DETECTOR RETROCESO PILOTO B5
"A01DDPLB6"	I 401.2	BOOL	// (A01E12) : DETECTOR RETROCESO PILOTO B6
"A01DDPLB7"	I 401.3	BOOL	// (A01E12) : DETECTOR RETROCESO PILOTO B7
"A01DEPLB4"	I 401.4	BOOL	// (A01E12) : DETECTOR AVANCE PILOTO B4
"A01DEPLB5"	I 401.5	BOOL	// (A01E12) : DETECTOR AVANCE PILOTO B5
"A01DEPLB6"	I 401.6	BOOL	// (A01E12) : DETECTOR AVANCE PILOTO B6
"A01DEPLB7"	I 401.7	BOOL	// (A01E12) : DETECTOR AVANCE PILOTO B7
"A01DDPLB8"	I 402.0	BOOL	// (A01E13) : DETECTOR RETROCESO PILOTO B8
"A01DDPLC1"	I 402.1	BOOL	// (A01E13) : DETECTOR RETROCESO PILOTO C1
"A01DDPLC2"	I 402.2	BOOL	// (A01E13) : DETECTOR RETROCESO PILOTO C2
"A01DDPLC3"	I 402.3	BOOL	// (A01E13) : DETECTOR RETROCESO PILOTO C3
"A01DEPLB8"	I 402.4	BOOL	// (A01E13) : DETECTOR AVANCE PILOTO B8
"A01DEPLC1"	I 402.5	BOOL	// (A01E13) : DETECTOR AVANCE PILOTO C1
"A01DEPLC2"	I 402.6	BOOL	// (A01E13) : DETECTOR AVANCE PILOTO C2
"A01DEPLC3"	I 402.7	BOOL	// (A01E13) : DETECTOR AVANCE PILOTO C3
"A01DDPLC4"	I 403.0	BOOL	// (A01E13) : DETECTOR RETROCESO PILOTO C4
"A01DDPLD1"	I 403.1	BOOL	// (A01E14) : DETECTOR RETROCESO PILOTO D1
"A01DDPLD2"	I 403.2	BOOL	// (A01E14) : DETECTOR RETROCESO PILOTO D2
"A01DDPLD3"	I 403.3	BOOL	// (A01E14) : DETECTOR RETROCESO PILOTO D3
"A01DEPLC4"	I 403.4	BOOL	// (A01E13) : DETECTOR AVANCE PILOTO C4
"A01DEPLD1"	I 403.5	BOOL	// (A01E14) : DETECTOR AVANCE PILOTO D1
"A01DEPLD2"	I 403.6	BOOL	// (A01E14) : DETECTOR AVANCE PILOTO D1
"A01DEPLD3"	I 403.7	BOOL	// (A01E14) : DETECTOR AVANCE PILOTO D3
"A01DDSRE1"	I 404.0	BOOL	// (A01E15) : DETECTOR RETROCESO APRIETE E1
"A01DDSRE2"	I 404.1	BOOL	// (A01E15) : DETECTOR RETROCESO APRIETE E2
"A01DDSRE3"	I 404.2	BOOL	// (A01E15) : DETECTOR RETROCESO APRIETE E3
"A01DDSRE4"	I 404.3	BOOL	// (A01E15) : DETECTOR RETROCESO APRIETE E4
"A01DESRE1"	I 404.4	BOOL	// (A01E15) : DETECTOR AVANCE APRIETE E1
"A01DESRE2"	I 404.5	BOOL	// (A01E15) : DETECTOR AVANCE APRIETE E2
"A01DESRE3"	I 404.6	BOOL	// (A01E15) : DETECTOR AVANCE APRIETE E3
"A01DESRE4"	I 404.7	BOOL	// (A01E15) : DETECTOR AVANCE APRIETE E4
"A01DDSRE5"	I 405.0	BOOL	// (A01E16) : DETECTOR RETROCESO APRIETE E5
"A01DDSRE6"	I 405.1	BOOL	// (A01E16) : DETECTOR RETROCESO APRIETE E6
"A01DDSRE7"	I 405.2	BOOL	// (A01E16) : DETECTOR RETROCESO APRIETE E7
"A01DDSRE8"	I 405.3	BOOL	// (A01E16) : DETECTOR RETROCESO APRIETE E8
"A01DESRE5"	I 405.4	BOOL	// (A01E16) : DETECTOR AVANCE APRIETE E5
"A01DESRE6"	I 405.5	BOOL	// (A01E16) : DETECTOR AVANCE APRIETE E6
"A01DESRE7"	I 405.6	BOOL	// (A01E16) : DETECTOR AVANCE APRIETE E7
"A01DESRE8"	I 405.7	BOOL	// (A01E16) : DETECTOR AVANCE APRIETE E8
"A01DDSRF1"	I 406.0	BOOL	// (A01E17) : DETECTOR RETROCESO APRIETE F1
"A01DDSRF2"	I 406.1	BOOL	// (A01E17) : DETECTOR RETROCESO APRIETE F2
"A01DDSRF3"	I 406.2	BOOL	// (A01E17) : DETECTOR RETROCESO APRIETE F3
"A01DDSRF4"	I 406.3	BOOL	// (A01E17) : DETECTOR RETROCESO APRIETE F4
"A01DESRF1"	I 406.4	BOOL	// (A01E17) : DETECTOR AVANCE APRIETE F1
"A01DESRF2"	I 406.5	BOOL	// (A01E17) : DETECTOR AVANCE APRIETE F2
"A01DESRF3"	I 406.6	BOOL	// (A01E17) : DETECTOR AVANCE APRIETE F3
"A01DESRF4"	I 406.7	BOOL	// (A01E17) : DETECTOR AVANCE APRIETE F4
"A01DDSRF5"	I 407.0	BOOL	// (A01E18) : DETECTOR RETROCESO APRIETE F5
"A01DDSRF6"	I 407.1	BOOL	// (A01E18) : DETECTOR RETROCESO APRIETE F6
"A01DDSRF7"	I 407.2	BOOL	// (A01E18) : DETECTOR RETROCESO APRIETE F7
"A01DDSRF8"	I 407.3	BOOL	// (A01E18) : DETECTOR RETROCESO APRIETE F8
"A01DESRF5"	I 407.4	BOOL	// (A01E18) : DETECTOR AVANCE APRIETE F5
"A01DESRF6"	I 407.5	BOOL	// (A01E18) : DETECTOR AVANCE APRIETE F6
"A01DESRF7"	I 407.6	BOOL	// (A01E18) : DETECTOR AVANCE APRIETE F7
"A01DESRF8"	I 407.7	BOOL	// (A01E18) : DETECTOR AVANCE APRIETE F8
"A01DDSRE9"	I 408.0	BOOL	// (A01E19) : DETECTOR RETROCESO APRIETE E9
"A01DDSRG2"	I 408.1	BOOL	// (A01E19) : DETECTOR RETROCESO APRIETE G2
"A01DDSRG3"	I 408.2	BOOL	// (A01E19) : DETECTOR RETROCESO APRIETE G3
"A01DDSRG4"	I 408.3	BOOL	// (A01E19) : DETECTOR RETROCESO APRIETE G4
"A01DESRE9"	I 408.4	BOOL	// (A01E19) : DETECTOR AVANCE APRIETE E9
"A01DESRG2"	I 408.5	BOOL	// (A01E19) : DETECTOR AVANCE APRIETE G2
"A01DESRG3"	I 408.6	BOOL	// (A01E19) : DETECTOR AVANCE APRIETE G3
"A01DESRG4"	I 408.7	BOOL	// (A01E19) : DETECTOR AVANCE APRIETE G4
"A01DDSRG5"	I 409.0	BOOL	// (A01E110) : DETECTOR RETROCESO APRIETE G5
"A01DDSRH1"	I 409.1	BOOL	// (A01E110) : DETECTOR RETROCESO APRIETE H1
"A01DDSRH2"	I 409.2	BOOL	// (A01E110) : DETECTOR RETROCESO APRIETE H2
"A01DDSRJ1"	I 409.3	BOOL	// (A01E110) : DETECTOR RETROCESO APRIETE J1
"A01DESRG5"	I 409.4	BOOL	// (A01E110) : DETECTOR AVANCE APRIETE G5
"A01DESRH1"	I 409.5	BOOL	// (A01E110) : DETECTOR AVANCE APRIETE H1
"A01DESRH2"	I 409.6	BOOL	// (A01E110) : DETECTOR AVANCE APRIETE H2
"A01DESRJ1"	I 409.7	BOOL	// (A01E110) : DETECTOR AVANCE APRIETE J1
"A01DDSRM1"	I 410.0	BOOL	// (A01E111) : DETECTOR RETROCESO APRIETE M1
"A01DDSRK2"	I 410.1	BOOL	// (A01E111) : DETECTOR RETROCESO APRIETE K2
"A01DDSRK3"	I 410.2	BOOL	// (A01E111) : DETECTOR RETROCESO APRIETE K3
"A01DDEJL1"	I 410.3	BOOL	// (A01E111) : DETECTOR RETROCESO EYECTOR L1
"A01DESRM1"	I 410.4	BOOL	// (A01E111) : DETECTOR AVANCE APRIETE M1
"A01DESRK2"	I 410.5	BOOL	// (A01E111) : DETECTOR AVANCE APRIETE K2
"A01DESRK3"	I 410.6	BOOL	// (A01E111) : DETECTOR AVANCE APRIETE K2
"A01DEEJL1"	I 410.7	BOOL	// (A01E111) : DETECTOR AVANCE EYECTOR L1
"A01DDEJL2"	I 411.0	BOOL	// (A01E112) : DETECTOR RETROCESO EYECTOR L2
"A01DDEJL3"	I 411.1	BOOL	// (A01E112) : DETECTOR RETROCESO EYECTOR L3
"A01DDEJL4"	I 411.2	BOOL	// (A01E112) : DETECTOR RETROCESO EYECTOR L4
"A01DDEJL5"	I 411.3	BOOL	// (A01E112) : DETECTOR RETROCESO EYECTOR L5
"A01DEEJL2"	I 411.4	BOOL	// (A01E112) : DETECTOR AVANCE EYECTOR L2
"A01DEEJL3"	I 411.5	BOOL	// (A01E112) : DETECTOR AVANCE EYECTOR L3
"A01DEEJL4"	I 411.6	BOOL	// (A01E112) : DETECTOR AVANCE EYECTOR L4
"A01DEEJL5"	I 411.7	BOOL	// (A01E112) : DETECTOR AVANCE EYECTOR L5
"A01DDEJL6"	I 412.0	BOOL	// (A01E113) : DETECTOR RETROCESO EYECTOR L6
"A01DDEJL7"	I 412.1	BOOL	// (A01E113) : DETECTOR RETROCESO EYECTOR L7
"A01DPP10"	I 412.2	BOOL	// (A01E114) : A01 PRESENCIA PIEZA DPP10
"A01DPP9"	I 412.3	BOOL	// (A01E114) : A01 PRESENCIA PIEZA DPP9
"A01DEEJL6"	I 412.4	BOOL	// (A01E113) : DETECTOR AVANCE EYECTOR L6
"A01DEEJL7"	I 412.5	BOOL	// (A01E113) : DETECTOR AVANCE EYECTOR L7
"SPARE412.6"	I 412.6	BOOL	// (A01E113) : RESERVE
"SPARE412.7"	I 412.7	BOOL	// (A01E113) : RESERVE
"A01DPP1"	I 413.0	BOOL	// (A01E114) : A01 PRESENCIA PIEZA DPP1
"A01DPP3"	I 413.1	BOOL	// (A01E114) : A01 PRESENCIA PIEZA DPP3
"A01DPP5"	I 413.2	BOOL	// (A01E114) : A01 PRESENCIA PIEZA DPP5
"A01DPP7"	I 413.3	BOOL	// (A01E114) : A01 PRESENCIA PIEZA DPP7
"A01DPP2"	I 413.4	BOOL	// (A01E114) : A01 PRESENCIA PIEZA DPP2
"A01DPP4"	I 413.5	BOOL	// (A01E114) : A01 PRESENCIA PIEZA DPP4
"A01DPP6"	I 413.6	BOOL	// (A01E114) : A01 PRESENCIA PIEZA DPP6
"A01DPP8"	I 413.7	BOOL	// (A01E114) : A01 PRESENCIA PIEZA DPP8
"SPARE414.0"	I 414.0	BOOL	// (A01E115) : RESERVE
"SPARE414.1"	I 414.1	BOOL	// (A01E115) : RESERVE
"SPARE414.2"	I 414.2	BOOL	// (A01E115) : RESERVE
"SPARE414.3"	I 414.3	BOOL	// (A01E115) : RESERVE
"SPARE414.4"	I 414.4	BOOL	// (A01E115) : RESERVE
"SPARE414.5"	I 414.5	BOOL	// (A01E115) : RESERVE
"SPARE414.6"	I 414.6	BOOL	// (A01E115) : RESERVE
"SPARE414.7"	I 414.7	BOOL	// (A01E115) : RESERVE
"B01DDPLA1"	I 460.0	BOOL	// (B01E11) : DETECTOR RETROCESO PILOTO A1
"B01DDPLA2"	I 460.1	BOOL	// (B01E11) : DETECTOR RETROCESO PILOTO A2
"B01DDPLA3"	I 460.2	BOOL	// (B01E11) : DETECTOR RETROCESO PILOTO A3
"B01DDPLA4"	I 460.3	BOOL	// (B01E11) : DETECTOR RETROCESO PILOTO A4
"B01DEPLA1"	I 460.4	BOOL	// (B01E11) : DETECTOR AVANCE PILOTO A1
"B01DEPLA2"	I 460.5	BOOL	// (B01E11) : DETECTOR AVANCE PILOTO A2
"B01DEPLA3"	I 460.6	BOOL	// (B01E11) : DETECTOR AVANCE PILOTO A3
"B01DEPLA4"	I 460.7	BOOL	// (B01E11) : DETECTOR AVANCE PILOTO A4
"B01DDPLA5"	I 461.0	BOOL	// (B01E12) : DETECTOR RETROCESO PILOTO A5
"B01DDPLA6"	I 461.1	BOOL	// (B01E12) : DETECTOR RETROCESO PILOTO A6
"B01DDSRB1"	I 461.2	BOOL	// (B01E12) : DETECTOR RETROCESO APRIETE B1
"B01DDSRB2"	I 461.3	BOOL	// (B01E12) : DETECTOR RETROCESO APRIETE B2
"B01DEPLA5"	I 461.4	BOOL	// (B01E12) : DETECTOR AVANCE PILOTO A5
"B01DEPLA6"	I 461.5	BOOL	// (B01E12) : DETECTOR AVANCE PILOTO A6
"B01DESRB1"	I 461.6	BOOL	// (B01E12) : DETECTOR AVANCE APRIETE B1
"B01DESRB2"	I 461.7	BOOL	// (B01E12) : DETECTOR AVANCE APRIETE B2
"B01DDPLC1"	I 462.0	BOOL	// (B01E13) : DETECTOR RETROCESO PILOTO C1
"B01DDPLD1"	I 462.1	BOOL	// (B01E13) : DETECTOR RETROCESO PILOTO D1
"B01DDPLA8"	I 462.2	BOOL	// (B01E13) : DETECTOR RETROCESO PILOTO A8
"B01DDPC"	I 462.3	BOOL	// (B01E13) : DETECTOR RETROCESO PILOTO PC
"B01DEPLC1"	I 462.4	BOOL	// (B01E13) : DETECTOR AVANCE PILOTO C1
"B01DEPLD1"	I 462.5	BOOL	// (B01E13) : DETECTOR AVANCE PILOTO D1
"B01DEPLA8"	I 462.6	BOOL	// (B01E13) : DETECTOR AVANCE PILOTO A8
"B01DEPC"	I 462.7	BOOL	// (B01E13) : DETECTOR AVANCE PILOTO PC
"B01DDPLD4"	I 463.0	BOOL	// (B01E14) : DETECTOR RETROCESO PILOTO D4
"B01DDPLD5"	I 463.1	BOOL	// (B01E14) : DETECTOR RETROCESO PILOTO D5
"B01DDSRF1"	I 463.2	BOOL	// (B01E14) : DETECTOR RETROCESO APRIETE F1
"B01DDSRF2"	I 463.3	BOOL	// (B01E15) : DETECTOR RETROCESO APRIETE F2
"B01DEPLD4"	I 463.4	BOOL	// (B01E14) : DETECTOR AVANCE PILOTO D4
"B01DEPLD5"	I 463.5	BOOL	// (B01E14) : DETECTOR AVANCE PILOTO D5
"B01DESRF1"	I 463.6	BOOL	// (B01E14) : DETECTOR AVANCE APRIETE F1
"B01DESRF2"	I 463.7	BOOL	// (B01E15) : DETECTOR AVANCE APRIETE F2
"B01DDSRG1"	I 464.0	BOOL	// (B01E15) : DETECTOR RETROCESO APRIETE G1
"B01DDSRG2"	I 464.1	BOOL	// (B01E15) : DETECTOR RETROCESO APRIETE G2
"B01DDSRG3"	I 464.2	BOOL	// (B01E15) : DETECTOR RETROCESO APRIETE G3
"B01DDSRG4"	I 464.3	BOOL	// (B01E15) : DETECTOR RETROCESO APRIETE G4
"B01DESRG1"	I 464.4	BOOL	// (B01E15) : DETECTOR AVANCE APRIETE G1
"B01DESRG2"	I 464.5	BOOL	// (B01E15) : DETECTOR AVANCE APRIETE G2
"B01DESRG3"	I 464.6	BOOL	// (B01E15) : DETECTOR AVANCE APRIETE G3
"B01DESRG4"	I 464.7	BOOL	// (B01E15) : DETECTOR AVANCE APRIETE G4
"B01DDSRG5"	I 465.0	BOOL	// (B01E16) : DETECTOR RETROCESO APRIETE G5
"B01DDSRG6"	I 465.1	BOOL	// (B01E16) : DETECTOR RETROCESO APRIETE G6
"B01DDSRH1"	I 465.2	BOOL	// (B01E16) : DETECTOR RETROCESO APRIETE H1
"B01DDSRH2"	I 465.3	BOOL	// (B01E16) : DETECTOR RETROCESO APRIETE H2
"B01DESRG5"	I 465.4	BOOL	// (B01E16) : DETECTOR AVANCE APRIETE G5
"B01DESRG6"	I 465.5	BOOL	// (B01E16) : DETECTOR AVANCE APRIETE G6
"B01DESRH1"	I 465.6	BOOL	// (B01E16) : DETECTOR AVANCE APRIETE H1
"B01DESRH2"	I 465.7	BOOL	// (B01E16) : DETECTOR AVANCE APRIETE H2
"B01DDSRH3"	I 466.0	BOOL	// (B01E17) : DETECTOR RETROCESO APRIETE H3
"B01DDSRH4"	I 466.1	BOOL	// (B01E17) : DETECTOR RETROCESO APRIETE H4
"B01DDSRH5"	I 466.2	BOOL	// (B01E17) : DETECTOR RETROCESO APRIETE H5
"B01DDSRH6"	I 466.3	BOOL	// (B01E17) : DETECTOR RETROCESO APRIETE H6
"B01DESRH3"	I 466.4	BOOL	// (B01E17) : DETECTOR AVANCE APRIETE H3
"B01DESRH4"	I 466.5	BOOL	// (B01E17) : DETECTOR AVANCE APRIETE H4
"B01DESRH5"	I 466.6	BOOL	// (B01E17) : DETECTOR AVANCE APRIETE H5
"B01DESRH6"	I 466.7	BOOL	// (B01E17) : DETECTOR AVANCE APRIETE H6
"B01DDSRJ1"	I 467.0	BOOL	// (B01E18) : DETECTOR RETROCESO APRIETE J1
"B01DDSRJ2"	I 467.1	BOOL	// (B01E18) : DETECTOR RETROCESO APRIETE J2
"B01DDSRJ3"	I 467.2	BOOL	// (B01E18) : DETECTOR RETROCESO APRIETE J3
"B01DDSRJ4"	I 467.3	BOOL	// (B01E18) : DETECTOR RETROCESO APRIETE J4
"B01DESRJ1"	I 467.4	BOOL	// (B01E18) : DETECTOR AVANCE APRIETE J1
"B01DESRJ2"	I 467.5	BOOL	// (B01E18) : DETECTOR AVANCE APRIETE J2
"B01DESRJ3"	I 467.6	BOOL	// (B01E18) : DETECTOR AVANCE APRIETE J3
"B01DESRJ4"	I 467.7	BOOL	// (B01E18) : DETECTOR AVANCE APRIETE J4
"B01DDSRJ5"	I 468.0	BOOL	// (B01E19) : DETECTOR RETROCESO APRIETE J5
"B01DDSRJ6"	I 468.1	BOOL	// (B01E19) : DETECTOR RETROCESO APRIETE J6
"B01DDEJK1"	I 468.2	BOOL	// (B01E19) : DETECTOR RETROCESO APRIETE K1
"B01DDEJK2"	I 468.3	BOOL	// (B01E19) : DETECTOR RETROCESO APRIETE K2
"B01DESRJ5"	I 468.4	BOOL	// (B01E19) : DETECTOR AVANCE APRIETE J5
"B01DESRJ6"	I 468.5	BOOL	// (B01E19) : DETECTOR AVANCE APRIETE J6
"B01DEEJK1"	I 468.6	BOOL	// (B01E19) : DETECTOR AVANCE APRIETE K1
"B01DEEJK2"	I 468.7	BOOL	// (B01E19) : DETECTOR AVANCE APRIETE K2
"B01DDEJK3"	I 469.0	BOOL	// (B01E110) : DETECTOR RETROCESO EYECTOR K3
"B01DDEJK4"	I 469.1	BOOL	// (B01E110) : DETECTOR RETROCESO EYECTOR K4
"B01DDEJK5"	I 469.2	BOOL	// (B01E110) : DETECTOR RETROCESO EYECTOR K5
"B01DDEJK6"	I 469.3	BOOL	// (B01E110) : DETECTOR RETROCESO EYECTOR K6
"B01DEEJK3"	I 469.4	BOOL	// (B01E110) : DETECTOR RETROCESO EYECTOR K3
"B01DEEJK4"	I 469.5	BOOL	// (B01E110) : DETECTOR RETROCESO EYECTOR K4
"B01DEEJK5"	I 469.6	BOOL	// (B01E110) : DETECTOR RETROCESO EYECTOR K5
"B01DEEJK6"	I 469.7	BOOL	// (B01E110) : DETECTOR RETROCESO EYECTOR K6
"B01DDEJK7"	I 470.0	BOOL	// (B01E111) : DETECTOR RETROCESO EYECTOR A7
"B01DDPLA7"	I 470.1	BOOL	// (B01E111) : DETECTOR RETROCESO PILOTO A7
"B01DDBM1"	I 470.3	BOOL	// (B01E111) : DETECTOR RETROCESO BRIDA MANUAL 1
"B01DEEJK7"	I 470.4	BOOL	// (B01E111) : DETECTOR AVANCE EYECTOR K7
"B01DEPLA7"	I 470.5	BOOL	// (B01E111) : DETECTOR AVANCE PILOTO A7
"B01DEBM1"	I 470.7	BOOL	// (B01E111) : DETECTOR AVANCE BRIDA MANUAL 1
"B01DPP1"	I 472.0	BOOL	// (B01E113) : B01 PRESENCIA PIEZA DPP1
"B01DPP3"	I 472.1	BOOL	// (B01E113) : B01 PRESENCIA PIEZA DPP3
"B01DPP5"	I 472.2	BOOL	// (B01E113) : B01 PRESENCIA PIEZA DPP5
"B01DPP7"	I 472.3	BOOL	// (B01E113) : B01 PRESENCIA PIEZA DPP3
"B01DPP2"	I 472.4	BOOL	// (B01E113) : B01 PRESENCIA PIEZA DPP2
"B01DPP4"	I 472.5	BOOL	// (B01E113) : B01 PRESENCIA PIEZA DPP4
"B01DPP6"	I 472.6	BOOL	// (B01E113) : B01 PRESENCIA PIEZA DPP6
"B01DPP8"	I 472.7	BOOL	// (B01E113) : B01 PRESENCIA PIEZA DPP8
"B01DPP9"	I 473.0	BOOL	// (B01E114) : B01 PRESENCIA PIEZA DPP9
"B01DPP10"	I 473.1	BOOL	// (B01E114) : B01 PRESENCIA PIEZA DPP10
"B01DPP11"	I 473.2	BOOL	// (B01E114) : B01 PRESENCIA PIEZA DPP11
"C01DEPLA1"	I 520.0	BOOL	// (C01E11) : DETECTOR RETROCESO PILOTO A1
"C01DEPLA2"	I 520.1	BOOL	// (C01E11) : DETECTOR RETROCESO PILOTO A2
"C01DEPLA3"	I 520.2	BOOL	// (C01E11) : DETECTOR RETROCESO PILOTO A3
"C01DDABB1"	I 520.3	BOOL	// (C01E11) : DETECTOR RETROCESO BATIENTE B1
"C01DDPLA1"	I 520.4	BOOL	// (C01E11) : DETECTOR AVANCE PILOTO A1
"C01DDPLA2"	I 520.5	BOOL	// (C01E11) : DETECTOR AVANCE PILOTO A2
"C01DDPLA3"	I 520.6	BOOL	// (C01E11) : DETECTOR AVANCE PILOTO A3
"C01DEABB1"	I 520.7	BOOL	// (C01E11) : DETECTOR AVANCE BATIENTE B1
"C01DDABB2"	I 521.0	BOOL	// (C01E12) : DETECTOR RETROCESO BATIENTE B2
"C01DDPLC1"	I 521.1	BOOL	// (C01E12) : DETECTOR RETROCESO PILOTO C1
"C01DDPLC2"	I 521.2	BOOL	// (C01E12) : DETECTOR RETROCESO PILOTO C2
"C01DDPLC3"	I 521.3	BOOL	// (C01E12) : DETECTOR RETROCESO PILOTO C3
"C01DEABB2"	I 521.4	BOOL	// (C01E12) : DETECTOR AVANCE BATIENTE B2
"C01DEPLC1"	I 521.5	BOOL	// (C01E12) : DETECTOR AVANCE PILOTO C1
"C01DEPLC2"	I 521.6	BOOL	// (C01E12) : DETECTOR AVANCE PILOTO C2
"C01DEPLC3"	I 521.7	BOOL	// (C01E12) : DETECTOR AVANCE PILOTO C3
"C01DDPLD1"	I 522.0	BOOL	// (C01E13) : DETECTOR RETROCESO PILOTO D1
"C01DDPLD2"	I 522.1	BOOL	// (C01E13) : DETECTOR RETROCESO PILOTO D2
"C01DDSRF1"	I 522.2	BOOL	// (C01E13) : DETECTOR RETROCESO APRIETE F1
"C01DDSRF2"	I 522.3	BOOL	// (C01E13) : DETECTOR RETROCESO APRIETE F2
"C01DEPLD1"	I 522.4	BOOL	// (C01E13) : DETECTOR AVANCE PILOTO D1
"C01DEPLD2"	I 522.5	BOOL	// (C01E13) : DETECTOR AVANCE PILOTO D2
"C01DESRF1"	I 522.6	BOOL	// (C01E13) : DETECTOR AVANCE APRIETE F1
"C01DESRF2"	I 522.7	BOOL	// (C01E13) : DETECTOR AVANCE APRIETE F2
"C01DDSRF3"	I 523.0	BOOL	// (C01E14) : DETECTOR RETROCESO APRIETE F3
"C01DDSRF4"	I 523.1	BOOL	// (C01E14) : DETECTOR RETROCESO APRIETE F4
"C01DDSRF5"	I 523.2	BOOL	// (C01E14) : DETECTOR RETROCESO APRIETE F5
"C01DESRF3"	I 523.4	BOOL	// (C01E14) : DETECTOR AVANCE APRIETE F3
"C01DESRF4"	I 523.5	BOOL	// (C01E14) : DETECTOR AVANCE APRIETE F4
"C01DESRF5"	I 523.6	BOOL	// (C01E14) : DETECTOR AVANCE APRIETE F5
"C01DDSRG1"	I 524.0	BOOL	// (C01E15) : DETECTOR RETROCESO APRIETE G1
"C01DDSRG2"	I 524.1	BOOL	// (C01E15) : DETECTOR RETROCESO APRIETE G2
"C01DDSRG3"	I 524.2	BOOL	// (C01E15) : DETECTOR RETROCESO APRIETE G3
"C01DDSRG4"	I 524.3	BOOL	// (C01E15) : DETECTOR RETROCESO APRIETE G4
"C01DESRG1"	I 524.4	BOOL	// (C01E15) : DETECTOR AVANCE APRIETE G1
"C01DESRG2"	I 524.5	BOOL	// (C01E15) : DETECTOR AVANCE APRIETE G2
"C01DESRG3"	I 524.6	BOOL	// (C01E15) : DETECTOR AVANCE APRIETE G3
"C01DESRG4"	I 524.7	BOOL	// (C01E15) : DETECTOR AVANCE APRIETE G4
"C01DDSRG5"	I 525.0	BOOL	// (C01E16) : DETECTOR RETROCESO APRIETE G5
"C01DDSRG6"	I 525.1	BOOL	// (C01E16) : DETECTOR RETROCESO APRIETE G6
"C01DDSRH1"	I 525.2	BOOL	// (C01E16) : DETECTOR RETROCESO APRIETE H1
"C01DDSRH2"	I 525.3	BOOL	// (C01E16) : DETECTOR RETROCESO APRIETE H2
"C01DESRG5"	I 525.4	BOOL	// (C01E16) : DETECTOR AVANCE APRIETE G5
"C01DESRG6"	I 525.5	BOOL	// (C01E16) : DETECTOR AVANCE APRIETE G6
"C01DESRH1"	I 525.6	BOOL	// (C01E16) : DETECTOR AVANCE APRIETE H1
"C01DESRH2"	I 525.7	BOOL	// (C01E16) : DETECTOR AVANCE APRIETE H2
"C01DDSRH3"	I 526.0	BOOL	// (C01E17) : DETECTOR RETROCESO APRIETE H3
"C01DDSRH4"	I 526.1	BOOL	// (C01E17) : DETECTOR RETROCESO APRIETE H4
"C01DDSRH5"	I 526.2	BOOL	// (C01E17) : DETECTOR RETROCESO APRIETE H5
"C01DDSRH6"	I 526.3	BOOL	// (C01E17) : DETECTOR RETROCESO APRIETE H6
"C01DESRH3"	I 526.4	BOOL	// (C01E17) : DETECTOR AVANCE APRIETE H3
"C01DESRH4"	I 526.5	BOOL	// (C01E17) : DETECTOR AVANCE APRIETE H4
"C01DESRH5"	I 526.6	BOOL	// (C01E17) : DETECTOR AVANCE APRIETE H5
"C01DESRH6"	I 526.7	BOOL	// (C01E17) : DETECTOR AVANCE APRIETE H6
"C01DDEJJ1"	I 527.0	BOOL	// (C01E18) : DETECTOR RETROCESO EYECTOR J1
"C01DDEJJ2"	I 527.1	BOOL	// (C01E18) : DETECTOR RETROCESO EYECTOR J2
"C01DDEJJ3"	I 527.2	BOOL	// (C01E18) : DETECTOR RETROCESO EYECTOR J3
"C01DDEJJ4"	I 527.3	BOOL	// (C01E18) : DETECTOR RETROCESO EYECTOR J4
"C01DEEJJ1"	I 527.4	BOOL	// (C01E18) : DETECTOR AVANCE EYECTOR J1
"C01DEEJJ2"	I 527.5	BOOL	// (C01E18) : DETECTOR AVANCE EYECTOR J2
"C01DEEJJ3"	I 527.6	BOOL	// (C01E18) : DETECTOR RETROCESO EYECTOR J3
"C01DEEJJ4"	I 527.7	BOOL	// (C01E18) : DETECTOR RETROCESO EYECTOR J4
"C01DDEJJ5"	I 528.0	BOOL	// (C01E19) : DETECTOR RETROCESO EYECTOR J5
"C01DDEJJ6"	I 528.1	BOOL	// (C01E19) : DETECTOR RETROCESO EYECTOR J6
"C01DDEJJ7"	I 528.2	BOOL	// (C01E19) : DETECTOR RETROCESO EYECTOR J7
"C01DEEJJ5"	I 528.4	BOOL	// (C01E19) : DETECTOR RETROCESO EYECTOR J5
"C01DEEJJ6"	I 528.5	BOOL	// (C01E19) : DETECTOR RETROCESO EYECTOR J6
"C01DEEJJ7"	I 528.6	BOOL	// (C01E19) : DETECTOR RETROCESO EYECTOR J7
"C01DPP1"	I 529.0	BOOL	// (C01E110) : C01 PRESENCIA PIEZA DPP1
"C01DPP3"	I 529.1	BOOL	// (C01E110) : C01 PRESENCIA PIEZA DPP3
"C01DPP4"	I 529.2	BOOL	// (C01E110) : C01 PRESENCIA PIEZA DPP4
"C01DPP2"	I 529.4	BOOL	// (C01E110) : C01 PRESENCIA PIEZA DPP2
"B02DDPLA1"	I 580.0	BOOL	// (B02E11) : DETECTOR RETROCESO PILOTO A1
"B02DDPLA2"	I 580.1	BOOL	// (B02E11) : DETECTOR RETROCESO PILOTO A2
"B02DDPLA3"	I 580.2	BOOL	// (B02E11) : DETECTOR RETROCESO PILOTO A3
"B02DDPLA4"	I 580.3	BOOL	// (B02E11) : DETECTOR RETROCESO PILOTO A4
"B02DEPLA1"	I 580.4	BOOL	// (B02E11) : DETECTOR AVANCE PILOTO A1
"B02DEPLA2"	I 580.5	BOOL	// (B02E11) : DETECTOR AVANCE PILOTO A2
"B02DEPLA3"	I 580.6	BOOL	// (B02E11) : DETECTOR AVANCE PILOTO A3
"B02DEPLA4"	I 580.7	BOOL	// (B02E11) : DETECTOR AVANCE PILOTO A4
"B02DDPLA5"	I 581.0	BOOL	// (B02E12) : DETECTOR RETROCESO PILOTO A5
"B02DDPLA6"	I 581.1	BOOL	// (B02E12) : DETECTOR RETROCESO PILOTO A6
"B02DDPLA7"	I 581.2	BOOL	// (B02E12) : DETECTOR RETROCESO PILOTO A7
"B02DDPLA8"	I 581.3	BOOL	// (B02E12) : DETECTOR RETROCESO PILOTO A8
"B02DEPLA5"	I 581.4	BOOL	// (B02E12) : DETECTOR AVANCE PILOTO A5
"B02DEPLA6"	I 581.5	BOOL	// (B02E12) : DETECTOR AVANCE PILOTO A6
"B02DEPLA7"	I 581.6	BOOL	// (B02E12) : DETECTOR AVANCE PILOTO A7
"B02DEPLA8"	I 581.7	BOOL	// (B02E12) : DETECTOR AVANCE PILOTO A8
"B02DDPLA9"	I 582.0	BOOL	// (B02E13) : DETECTOR RETROCESO PILOTO A9
"B02DESRB1"	I 582.1	BOOL	// (B02E13) : DETECTOR RETROCESO APRIETE B1
"B02DESRB2"	I 582.2	BOOL	// (B02E13) : DETECTOR RETROCESO APRIETE B2
"B02DDPLC1"	I 582.3	BOOL	// (B02E13) : DETECTOR RETROCESO PILOTO C1
"B02DEPLA9"	I 582.4	BOOL	// (B02E13) : DETECTOR AVANCE PILOTO A9
"B02DDSRB1"	I 582.5	BOOL	// (B02E13) : DETECTOR AVANCE APRIETE B1
"B02DDSRB2"	I 582.6	BOOL	// (B02E13) : DETECTOR AVANCE APRIETE B2
"B02DEPLC1"	I 582.7	BOOL	// (B02E13) : DETECTOR AVANCE PILOTO C1
"B02DDPLD1"	I 583.0	BOOL	// (B02E14) : DETECTOR RETROCESO PILOTO D1
"B02DDPLD2"	I 583.1	BOOL	// (B02E14) : DETECTOR RETROCESO PILOTO D2
"B02DDSRF1"	I 583.2	BOOL	// (B02E14) : DETECTOR RETROCESO APRIETE F1
"B02DDSRF2"	I 583.3	BOOL	// (B02E14) : DETECTOR RETROCESO APRIETE F2
"B02DEPLD1"	I 583.4	BOOL	// (B02E14) : DETECTOR AVANCE PILOTO D1
"B02DEPLD2"	I 583.5	BOOL	// (B02E14) : DETECTOR AVANCE PILOTO D2
"B02DESRF1"	I 583.6	BOOL	// (B02E14) : DETECTOR AVANCE APRIETE F1
"B02DESRF2"	I 583.7	BOOL	// (B02E14) : DETECTOR AVANCE APRIETE F2
"B02DDSRG1"	I 584.0	BOOL	// (B02E15) : DETECTOR RETROCESO APRIETE G1
"B02DDSRG2"	I 584.1	BOOL	// (B02E15) : DETECTOR RETROCESO PILOTO G2 (RH)
"B02DDSRG3"	I 584.2	BOOL	// (B02E15) : DETECTOR RETROCESO PILOTO G3 (RH)
"B02DSD1"	I 584.3	BOOL	// (B02E15) : DETECTOR SENSOR  DIVERSIDAD 1
"B02DESRG1"	I 584.4	BOOL	// (B02E15) : DETECTOR AVANCE APRIETE G1
"B02DESRG2"	I 584.5	BOOL	// (B02E15) : DETECTOR AVANCE PILOTO G2 (RH)
"B02DESRG3"	I 584.6	BOOL	// (B02E15) : DETECTOR AVANCE PILOTO G3 (RH)
"B02DDSRH1"	I 585.0	BOOL	// (B02E16) : DETECTOR RETROCESO APRIETE H1
"B02DDSRH2"	I 585.1	BOOL	// (B02E16) : DETECTOR RETROCESO APRIETE H2
"B02DDSRH3"	I 585.2	BOOL	// (B02E16) : DETECTOR RETROCESO APRIETE H3
"B02DDSRH4"	I 585.3	BOOL	// (B02E16) : DETECTOR RETROCESO APRIETE H4
"B02DESRH1"	I 585.4	BOOL	// (B02E16) : DETECTOR AVANCE APRIETE H1
"B02DESRH2"	I 585.5	BOOL	// (B02E16) : DETECTOR AVANCE APRIETE H2
"B02DESRH3"	I 585.6	BOOL	// (B02E16) : DETECTOR AVANCE APRIETE H3
"B02DESRH4"	I 585.7	BOOL	// (B02E16) : DETECTOR AVANCE APRIETE H4
"B02DDSRH5"	I 586.0	BOOL	// (B02E17) : DETECTOR RETROCESO APRIETE H5
"B02DDSRJ1"	I 586.1	BOOL	// (B02E17) : DETECTOR RETROCESO APRIETE J1
"B02DDSRJ2"	I 586.2	BOOL	// (B02E17) : DETECTOR RETROCESO APRIETE J2
"B02DDSRJ3"	I 586.3	BOOL	// (B02E17) : DETECTOR RETROCESO APRIETE J3
"B02DESRH5"	I 586.4	BOOL	// (B02E17) : DETECTOR AVANCE APRIETE H5
"B02DESRJ1"	I 586.5	BOOL	// (B02E17) : DETECTOR AVANCE APRIETE J1
"B02DESRJ2"	I 586.6	BOOL	// (B02E17) : DETECTOR AVANCE APRIETE J2
"B02DESRJ3"	I 586.7	BOOL	// (B02E17) : DETECTOR AVANCE APRIETE J3
"B02DDSRJ4"	I 587.0	BOOL	// (B02E18) : DETECTOR RETROCESO APRIETE J4
"B02DDSRJ5"	I 587.1	BOOL	// (B02E18) : DETECTOR RETROCESO APRIETE J5
"B02DDSRJ6"	I 587.2	BOOL	// (B02E18) : DETECTOR RETROCESO APRIETE J6
"B02DESRJ4"	I 587.4	BOOL	// (B02E18) : DETECTOR AVANCE APRIETE J4
"B02DESRJ5"	I 587.5	BOOL	// (B02E18) : DETECTOR AVANCE APRIETE J5
"B02DESRJ6"	I 587.6	BOOL	// (B02E18) : DETECTOR AVANCE APRIETE J6
"B02DDSRK1"	I 588.0	BOOL	// (B02E19) : DETECTOR RETROCESO APRIETE K1
"B02DDSRK2"	I 588.1	BOOL	// (B02E19) : DETECTOR RETROCESO APRIETE K2
"B02DDSRK3"	I 588.2	BOOL	// (B02E19) : DETECTOR RETROCESO APRIETE K3
"B02DDSRK4"	I 588.3	BOOL	// (B02E19) : DETECTOR RETROCESO APRIETE K4
"B02DESRK1"	I 588.4	BOOL	// (B02E19) : DETECTOR AVANCE APRIETE K1
"B02DESRK2"	I 588.5	BOOL	// (B02E19) : DETECTOR AVANCE APRIETE K2
"B02DESRK3"	I 588.6	BOOL	// (B02E19) : DETECTOR AVANCE APRIETE K3
"B02DESRK4"	I 588.7	BOOL	// (B02E19) : DETECTOR AVANCE APRIETE K4
"B02DDSRK5"	I 589.0	BOOL	// (B02E110) : DETECTOR RETROCESO APRIETE K5
"B02DDSRK6"	I 589.1	BOOL	// (B02E110) : DETECTOR RETROCESO APRIETE K6
"B02DDSRK7"	I 589.2	BOOL	// (B02E110) : DETECTOR RETROCESO APRIETE K7
"B02DDSRK8"	I 589.3	BOOL	// (B02E110) : DETECTOR RETROCESO APRIETE K8
"B02DESRK5"	I 589.4	BOOL	// (B02E110) : DETECTOR AVANCE APRIETE K5
"B02DESRK6"	I 589.5	BOOL	// (B02E110) : DETECTOR AVANCE APRIETE K6
"B02DESRK7"	I 589.6	BOOL	// (B02E110) : DETECTOR AVANCE APRIETE K7
"B02DESRK8"	I 589.7	BOOL	// (B02E110) : DETECTOR AVANCE APRIETE K8
"B02DDEJL1"	I 590.0	BOOL	// (B02E111) : DETECTOR RETROCESO EYECTOR L1
"B02DDEJL2"	I 590.1	BOOL	// (B02E111) : DETECTOR RETROCESO EYECTOR L2
"B02DDEJL3"	I 590.2	BOOL	// (B02E111) : DETECTOR RETROCESO EYECTOR L3
"B02DDEJL4"	I 590.3	BOOL	// (B02E111) : DETECTOR RETROCESO EYECTOR L4
"B02DEEJL1"	I 590.4	BOOL	// (B02E111) : DETECTOR AVANCE EYECTOR L1
"B02DEEJL2"	I 590.5	BOOL	// (B02E111) : DETECTOR AVANCE EYECTOR L2
"B02DEEJL3"	I 590.6	BOOL	// (B02E111) : DETECTOR AVANCE EYECTOR L3
"B02DEEJL4"	I 590.7	BOOL	// (B02E111) : DETECTOR AVANCE EYECTOR L4
"B02DDEJL5"	I 591.0	BOOL	// (B02E112) : DETECTOR RETROCESO EYECTOR L5
"B02DDEJL6"	I 591.1	BOOL	// (B02E112) : DETECTOR RETROCESO EYECTOR L6
"B02DDEJL7"	I 591.2	BOOL	// (B02E112) : DETECTOR RETROCESO EYECTOR L7
"B02DEEJL5"	I 591.4	BOOL	// (B02E112) : DETECTOR AVANCE EYECTOR L5
"B02DEEJL6"	I 591.5	BOOL	// (B02E112) : DETECTOR AVANCE EYECTOR L6
"B02DEEJL7"	I 591.6	BOOL	// (B02E112) : DETECTOR AVANCE EYECTOR L7
"B02DPP1"	I 592.0	BOOL	// (B02E113) : B02 PRESENCIA PIEZA DPP1
"B02DPP3"	I 592.1	BOOL	// (B02E113) : B02 PRESENCIA PIEZA DPP3
"B02DPP5"	I 592.2	BOOL	// (B02E113) : B02 PRESENCIA PIEZA DPP5
"B02DPP7"	I 592.3	BOOL	// (B02E113) : B02 PRESENCIA PIEZA DPP7
"B02DPP2"	I 592.4	BOOL	// (B02E113) : B02 PRESENCIA PIEZA DPP2
"B02DPP4"	I 592.5	BOOL	// (B02E113) : B02 PRESENCIA PIEZA DPP4
"B02DPP6"	I 592.6	BOOL	// (B02E113) : B02 PRESENCIA PIEZA DPP6
"B02DPP8"	I 592.7	BOOL	// (B02E113) : B02 PRESENCIA PIEZA DPP8
"B02DPP9"	I 593.0	BOOL	// (B02E113) : B02 PRESENCIA PIEZA DPP9
"B02DPP11"	I 593.1	BOOL	// (B02E113) : B02 PRESENCIA PIEZA DPP11
"B02DPP10"	I 593.4	BOOL	// (B02E113) : B02 PRESENCIA PIEZA DPP10
"C02DDPLA1"	I 640.0	BOOL	// (C02E11) : DETECTOR RETROCESO PILOTO A1
"C02DDPLA2"	I 640.1	BOOL	// (C02E11) : DETECTOR RETROCESO PILOTO A2
"C02DDPLA3"	I 640.2	BOOL	// (C02E11) : DETECTOR RETROCESO PILOTO A3
"C02DDABB1"	I 640.3	BOOL	// (C02E11) : DETECTOR RETROCESO BATIENTE B1
"C02DEPLA1"	I 640.4	BOOL	// (C02E11) : DETECTOR AVANCE PILOTO A1
"C02DEPLA2"	I 640.5	BOOL	// (C02E11) : DETECTOR AVANCE PILOTO A2
"C02DEPLA3"	I 640.6	BOOL	// (C02E11) : DETECTOR AVANCE PILOTO A3
"C02DEABB1"	I 640.7	BOOL	// (C02E11) : DETECTOR AVANCE BATIENTE B1
"C02DDABB2"	I 641.0	BOOL	// (C02E12) : DETECTOR RETROCESO BATIENTE B2
"C02DDABB3"	I 641.1	BOOL	// (C02E12) : DETECTOR RETROCESO BATIENTE B3
"C02DDABB4"	I 641.2	BOOL	// (C02E12) : DETECTOR RETROCESO BATIENTE B4
"C02DDABB5"	I 641.3	BOOL	// (C02E12) : DETECTOR RETROCESO BATIENTE B5
"C02DEABB2"	I 641.4	BOOL	// (C02E12) : DETECTOR AVANCE BATIENTE B2
"C02DEABB3"	I 641.5	BOOL	// (C02E12) : DETECTOR AVANCE BATIENTE B3
"C02DEABB4"	I 641.6	BOOL	// (C02E12) : DETECTOR AVANCE BATIENTE B4
"C02DEABB5"	I 641.7	BOOL	// (C02E12) : DETECTOR AVANCE BATIENTE B5
"C02DDABB6"	I 642.0	BOOL	// (C02E13) : DETECTOR RETROCESO BATIENTE B6
"C02DDABB7"	I 642.1	BOOL	// (C02E13) : DETECTOR RETROCESO BATIENTE B7
"C02DDPLC1"	I 642.2	BOOL	// (C02E13) : DETECTOR RETROCESO PILOTO C1
"C02DDPLC2"	I 642.3	BOOL	// (C02E13) : DETECTOR RETROCESO PILOTO C2
"C02DEABB6"	I 642.4	BOOL	// (C02E13) : DETECTOR AVANCE BATIENTE B6
"C02DEABB7"	I 642.5	BOOL	// (C02E13) : DETECTOR AVANCE BATIENTE B7
"C02DEPLC1"	I 642.6	BOOL	// (C02E13) : DETECTOR AVANCE PILOTO C1
"C02DEPLC2"	I 642.7	BOOL	// (C02E13) : DETECTOR AVANCE PILOTO C2
"C02DDSRE1"	I 643.0	BOOL	// (C02E14) : DETECTOR RETROCESO APRIETE E1
"C02DDSRE2"	I 643.1	BOOL	// (C02E14) : DETECTOR RETROCESO APRIETE E2
"C02DDSRF1"	I 643.2	BOOL	// (C02E14) : DETECTOR RETROCESO APRIETE F1
"C02DDSRF2"	I 643.3	BOOL	// (C02E14) : DETECTOR RETROCESO APRIETE F2
"C02DESRE1"	I 643.4	BOOL	// (C02E14) : DETECTOR AVANCE APRIETE E1
"C02DESRE2"	I 643.5	BOOL	// (C02E14) : DETECTOR AVANCE APRIETE E2
"C02DESRF1"	I 643.6	BOOL	// (C02E14) : DETECTOR AVANCE APRIETE F1
"C02DESRF2"	I 643.7	BOOL	// (C02E14) : DETECTOR AVANCE APRIETE F2
"C02DDSRF3"	I 644.0	BOOL	// (C02E15) : DETECTOR RETROCESO APRIETE F3
"C02DDSRF4"	I 644.1	BOOL	// (C02E15) : DETECTOR RETROCESO APRIETE F4
"C02DDSRF5"	I 644.2	BOOL	// (C02E15) : DETECTOR RETROCESO APRIETE F5
"C02DDSRF6"	I 644.3	BOOL	// (C02E15) : DETECTOR RETROCESO APRIETE F6
"C02DESRF3"	I 644.4	BOOL	// (C02E15) : DETECTOR AVANCE APRIETE F3
"C02DESRF4"	I 644.5	BOOL	// (C02E15) : DETECTOR AVANCE APRIETE F4
"C02DESRF5"	I 644.6	BOOL	// (C02E15) : DETECTOR AVANCE APRIETE F5
"C02DESRF6"	I 644.7	BOOL	// (C02E15) : DETECTOR AVANCE APRIETE F6
"C02DDSRF7"	I 645.0	BOOL	// (C02E16) : DETECTOR RETROCESO APRIETE F7
"C02DDSRG1"	I 645.1	BOOL	// (C02E16) : DETECTOR RETROCESO APRIETE G1
"C02DDSRG2"	I 645.2	BOOL	// (C02E16) : DETECTOR RETROCESO APRIETE G2
"C02DDSRG3"	I 645.3	BOOL	// (C02E16) : DETECTOR RETROCESO APRIETE G3
"C02DESRF7"	I 645.4	BOOL	// (C02E16) : DETECTOR AVANCE APRIETE F7
"C02DESRG1"	I 645.5	BOOL	// (C02E16) : DETECTOR AVANCE APRIETE G1
"C02DESRG2"	I 645.6	BOOL	// (C02E16) : DETECTOR AVANCE APRIETE G2
"C02DESRG3"	I 645.7	BOOL	// (C02E16) : DETECTOR AVANCE APRIETE G3
"C02DDSRG4"	I 646.0	BOOL	// (C02E17) : DETECTOR RETROCESO APRIETE G4
"C02DDSRG5"	I 646.1	BOOL	// (C02E17) : DETECTOR RETROCESO APRIETE G5
"C02DDSRH1"	I 646.2	BOOL	// (C02E17) : DETECTOR RETROCESO APRIETE H1
"C02DDSRH2"	I 646.3	BOOL	// (C02E17) : DETECTOR RETROCESO APRIETE H2
"C02DESRG4"	I 646.4	BOOL	// (C02E17) : DETECTOR AVANCE APRIETE G4
"C02DESRG5"	I 646.5	BOOL	// (C02E17) : DETECTOR AVANCE APRIETE G5
"C02DESRH1"	I 646.6	BOOL	// (C02E17) : DETECTOR AVANCE APRIETE H1
"C02DESRH2"	I 646.7	BOOL	// (C02E17) : DETECTOR AVANCE APRIETE H2
"C02DDSRH3"	I 647.0	BOOL	// (C02E18) : DETECTOR RETROCESO APRIETE H3
"C02DDSRH4"	I 647.1	BOOL	// (C02E18) : DETECTOR RETROCESO APRIETE H4
"C02DDSRH5"	I 647.2	BOOL	// (C02E18) : DETECTOR RETROCESO APRIETE H5
"C02DESRH3"	I 647.4	BOOL	// (C02E18) : DETECTOR AVANCE APRIETE H3
"C02DESRH4"	I 647.5	BOOL	// (C02E18) : DETECTOR AVANCE APRIETE H4
"C02DESRH5"	I 647.6	BOOL	// (C02E18) : DETECTOR AVANCE APRIETE H5
"C02DDEJJ1"	I 648.0	BOOL	// (C02E19) : DETECTOR RETROCESO EYECTOR J1
"C02DDEJJ2"	I 648.1	BOOL	// (C02E19) : DETECTOR RETROCESO EYECTOR J2
"C02DDEJJ3"	I 648.2	BOOL	// (C02E19) : DETECTOR RETROCESO EYECTOR J3
"C02DDEJJ4"	I 648.3	BOOL	// (C02E19) : DETECTOR RETROCESO EYECTOR J4
"C02DEEJJ1"	I 648.4	BOOL	// (C02E19) : DETECTOR AVANCE EYECTOR J1
"C02DEEJJ2"	I 648.5	BOOL	// (C02E19) : DETECTOR AVANCE EYECTOR J2
"C02DEEJJ3"	I 648.6	BOOL	// (C02E19) : DETECTOR AVANCE EYECTOR J3
"C02DEEJJ4"	I 648.7	BOOL	// (C02E19) : DETECTOR AVANCE EYECTOR J4
"C02DDEJJ5"	I 649.0	BOOL	// (C02E110) : DETECTOR RETROCESO EYECTOR J5
"C02DDEJJ6"	I 649.1	BOOL	// (C02E110) : DETECTOR RETROCESO EYECTOR J6
"C02DDEJJ7"	I 649.2	BOOL	// (C02E110) : DETECTOR RETROCESO EYECTOR J7
"C02DEEJJ5"	I 649.4	BOOL	// (C02E110) : DETECTOR AVANCE EYECTOR J5
"C02DEEJJ6"	I 649.5	BOOL	// (C02E110) : DETECTOR AVANCE EYECTOR J6
"C02DEEJJ7"	I 649.6	BOOL	// (C02E110) : DETECTOR AVANCE EYECTOR J7
"C02DPP1"	I 650.0	BOOL	// (C02E111) : C02 PART PRESENT DPP1
"C02DPP3"	I 650.1	BOOL	// (C02E111) : C02 PART PRESENT DPP3
"C02DPP2"	I 650.4	BOOL	// (C02E111) : C02 PART PRESENT DPP2
"C02DPP4"	I 650.5	BOOL	// (C02E111) : C02 PART PRESENT DPP4
"BA0"	M 0.0	BOOL	// FACILITY: BIT ALWAYS OFF / ILOT: BIT TOUJOURS A 0
"BA1"	M 0.1	BOOL	// FACILITY: BIT ALWAYS ON / ILOT: BIT TOUJOURS A 1
"BA1LIEN"	M 0.2	BOOL	// FACILITY: BIT ALWAYS ON (LINK IN THE PROGRAMMING NETWORK)
"SHUNT"	M 0.3	BOOL	// BIT FOR BYPASS DURING FACILITY START UP / BIT SHUNT POUR LA MISE AU POINT
"PERSO"	M 0.4	BOOL	// NEED TO PERSONALIZE BY THE PROGRAMMER / EQUATION A PERSONNALISER
"POUB"	M 0.5	BOOL	// DUST BIN BIT / BIT POUBELLE
"SYSFROID"	M 0.7	BOOL	// DETECTING COLD START PLC (OB102) / DETECTION DEMARRAGE A FROID API (OB102)
"ICL080S"	M 1.4	BOOL
"ICL2S"	M 1.7	BOOL
"shunt_test"	M 5.0	BOOL
"IADF"	M 10.1	BOOL	// FACILITY: FAULT RESET INFORMATION (SAFETY)
"IR"	M 10.2	BOOL	// FACILITY: CONTROL ON INFORMATION (SAFETY)
"ANUL_X_PRUEBA"	M 10.4	BOOL	// PARA PRUEBAS DANIEL
"CDC_D"	M 10.5	BOOL	// BIT ESPECIAL PARA LADO DERECHA
"RepRecalL38"	M 10.6	BOOL	// Reponse automatique a une demande d'injection L38 (provisoire)
"ANULADO"	M 10.7	BOOL	// Bit para anulacion sensado mov. Pedidos por Geometras
"Z1DEF_MAJ"	M 11.0	BOOL	// ZONA 1: MAJOR FAULT (SAFETY)
"Z1IADF"	M 11.1	BOOL	// ZONA 1: FAULT RESET INFORMATION (SAFETY)
"Z1IR"	M 11.2	BOOL	// ZONA 1: CONTROL ON INFORMATION (SAFETY)
"Z1IAFJ"	M 11.3	BOOL	// ZONA 1: END OF PRODUCTION STOP INFORMATION (SAFETY)
"Z1MAUTO"	M 11.4	BOOL	// ZONA 1: ZONA EN MODO AUTOMATIC (SAFETY)
"Z1MDV"	M 11.5	BOOL	// ZONA 1: ZONA EN DEVERMINAGE
"Z1SLDEV"	M 11.6	BOOL	// ZONA 1: PULSADOR DEVERMINAGE
"DEFMAJ_AU_ES"	M 11.7	BOOL	// ZONA 1: INHIBICION DEFECTO SECURIDAD AU / ES
"A01.DEF"	M 20.0	BOOL	// DEFECTO GENERAL DE MESA A01
"B01.DEF"	M 20.1	BOOL	// DEFECTO GENERAL DE MESA B01
"C01.DEF"	M 20.2	BOOL	// DEFECTO GENERAL DE LA MESA C01
"B02.DEF"	M 20.3	BOOL	// DEFECTO GENERAL MESA B02
"C02.DEF"	M 20.4	BOOL	// DEFECTO GENERAL MESA C02
"xAlas"	M 30.0	BOOL
"A01"	M 30.1	BOOL
"SHUNT_VAL_X52"	M 77.4	BOOL
"Transferencia A0 a A0W"	M 200.0	BOOL	// Transferencia de palabra desde A0 a A0W OK
"A01_AT_A11"	M 201.0	BOOL	// A0: OPERATOR A1 WORK AUTORIZATION / AUTORIZACION DE TRABAJO OPERARIO A1
"A01_ET_A11"	M 201.1	BOOL	// A0: OPERATOR A1 WORK AUTORIZATION / AUTORIZACION DE TRABAJO OPERARIO A1
"A01_AT_A12"	M 202.0	BOOL	// A0: OPERATOR A2 WORK AUTORIZATION / AUTORIZACION DE TRABAJO OPERARIO A2
"A01_ET_A12"	M 202.1	BOOL	// A0: OPERATOR A2 WORK AUTORIZATION / AUTORIZACION DE TRABAJO OPERARIO A2
"B01_AT_B11"	M 203.0	BOOL	// A0: OPERATOR A3 WORK AUTORIZATION / AUTORIZACION DE TRABAJO OPERARIO A3
"B01_ET_B11"	M 203.1	BOOL	// A0: OPERATOR A3 WORK AUTORIZATION / AUTORIZACION DE TRABAJO OPERARIO A3
"B01_AT_B12"	M 204.0	BOOL	// B0: OPERATOR B1 WORK AUTORIZATION / AUTORIZACION DE TRABAJO OPERARIO B1
"B01_ET_B12"	M 204.1	BOOL	// B0: OPERATOR B1 WORK AUTORIZATION / AUTORIZACION DE TRABAJO OPERARIO B1
"B01_AT_B13"	M 204.2	BOOL	// B0: OPERATOR B2 WORK AUTORIZATION / AUTORIZACION DE TRABAJO OPERARIO B2
"B01_ET_B13"	M 204.3	BOOL	// B0: OPERATOR B1 WORK AUTORIZATION / AUTORIZACION DE TRABAJO OPERARIO B1
"C01_AT_C11"	M 205.0	BOOL	// C0: OPERATOR C1 WORK AUTORIZATION / AUTORIZACION DE TRABAJO OPERARIO C1
"C01_ET_C11"	M 205.1	BOOL	// C0: OPERATOR C1 WORK AUTORIZATION / AUTORIZACION DE TRABAJO OPERARIO C1
"C01_AT_C12"	M 205.2	BOOL	// C0: OPERATOR C1 WORK AUTORIZATION / AUTORIZACION DE TRABAJO OPERARIO C1
"C01_ET_C12"	M 205.3	BOOL	// C0: OPERATOR C1 WORK AUTORIZATION / AUTORIZACION DE TRABAJO OPERARIO C1
"C01_AT_C13"	M 205.4	BOOL	// C0: OPERATOR C1 WORK AUTORIZATION / AUTORIZACION DE TRABAJO OPERARIO C1
"C01_ET_C13"	M 205.5	BOOL	// C0: OPERATOR C1 WORK AUTORIZATION / AUTORIZACION DE TRABAJO OPERARIO C1
"B02_AT_B21"	M 205.6	BOOL	// A0: OPERATOR A3 WORK AUTORIZATION / AUTORIZACION DE TRABAJO OPERARIO A3
"B02_ET_B21"	M 205.7	BOOL	// A0: OPERATOR A3 WORK AUTORIZATION / AUTORIZACION DE TRABAJO OPERARIO A3
"B02_AT_B22"	M 206.0	BOOL	// B0: OPERATOR B1 WORK AUTORIZATION / AUTORIZACION DE TRABAJO OPERARIO B1
"B02_ET_B22"	M 206.1	BOOL	// B0: OPERATOR B1 WORK AUTORIZATION / AUTORIZACION DE TRABAJO OPERARIO B1
"B02_AT_B23"	M 206.2	BOOL	// B0: OPERATOR B2 WORK AUTORIZATION / AUTORIZACION DE TRABAJO OPERARIO B2
"B02_ET_B23"	M 206.3	BOOL	// B0: OPERATOR B1 WORK AUTORIZATION / AUTORIZACION DE TRABAJO OPERARIO B1
"C02_AT_C21"	M 206.4	BOOL	// C0: OPERATOR C1 WORK AUTORIZATION / AUTORIZACION DE TRABAJO OPERARIO C1
"C02_ET_C21"	M 206.5	BOOL	// C0: OPERATOR C1 WORK AUTORIZATION / AUTORIZACION DE TRABAJO OPERARIO C1
"C02_AT_C22"	M 206.6	BOOL	// C0: OPERATOR C1 WORK AUTORIZATION / AUTORIZACION DE TRABAJO OPERARIO C1
"C02_ET_C22"	M 206.7	BOOL	// C0: OPERATOR C1 WORK AUTORIZATION / AUTORIZACION DE TRABAJO OPERARIO C1
"C02_AT_C23"	M 207.0	BOOL	// C0: OPERATOR C1 WORK AUTORIZATION / AUTORIZACION DE TRABAJO OPERARIO C1
"C02_ET_C23"	M 207.1	BOOL	// C0: OPERATOR C1 WORK AUTORIZATION / AUTORIZACION DE TRABAJO OPERARIO C1
"A11SOPVINH"	M 300.0	BOOL	// A11 LAMPADA SECURIDAD INACTIVO
"A12SOPVINH"	M 300.1	BOOL	// A12 LAMPADA SECURIDAD INACTIVO
"B11SOPVINH"	M 300.2	BOOL	// B11 LAMPADA SECURIDAD INACTIVO
"B12SOPVINH"	M 300.3	BOOL	// B12 LAMPADA SECURIDAD INACTIVO
"B13SOPVINH"	M 300.4	BOOL	// B13 LAMPADA SECURIDAD INACTIVO
"B21SOPVINH"	M 300.5	BOOL	// B21 LAMPADA SECURIDAD INACTIVO
"B22SOPVINH"	M 300.6	BOOL	// B22 LAMPADA SECURIDAD INACTIVO
"B23SOPVINH"	M 300.7	BOOL	// B23 LAMPADA SECURIDAD INACTIVO
"C11SOPVINH"	M 301.0	BOOL	// C11 LAMPADA SECURIDAD INACTIVO
"C12SOPVINH"	M 301.1	BOOL	// C12 LAMPADA SECURIDAD INACTIVO
"C13SOPVINH"	M 301.2	BOOL	// C13 LAMPADA SECURIDAD INACTIVO
"C21SOPVINH"	M 301.3	BOOL	// C21 LAMPADA SECURIDAD INACTIVO
"C22SOPVINH"	M 301.4	BOOL	// C22 LAMPADA SECURIDAD INACTIVO
"C23SOPVINH"	M 301.5	BOOL	// C23 LAMPADA SECURIDAD INACTIVO
"A01XEDPLB"	M 400.0	BOOL	// A01 AUXILIAR EV. RETROCESO PILOTO B
"A01XEEPLB"	M 400.1	BOOL	// A01 AUXILIAR  EV. AVANCE PILOTO B
"B01XEDPLA"	M 400.2	BOOL	// B01 AUXILIAR EV. RETROCESO PILOTO A
"B01XEEPLA"	M 400.3	BOOL	// B01 AUXILIAR  EV. AVANCE PILOTO A
"B02XEDPLA"	M 400.4	BOOL	// B01 AUXILIAR EV. RETROCESO PILOTO A
"B02XEEPLA"	M 400.5	BOOL	// B01 AUXILIAR  EV. AVANCE PILOTO A
"C01XEDPLA"	M 400.6	BOOL	// C01 AUXILIAR EV. RETROCESO PILOTO A
"C01XEEPLA"	M 400.7	BOOL	// C01 AUXILIAR  EV. AVANCE PILOTO A
"C02XEDPLA"	M 401.0	BOOL	// C02 AUXILIAR EV. RETROCESO PILOTO A
"C02XEEPLA"	M 401.2	BOOL	// C02 AUXILIAR  EV. AVANCE PILOTO A
"C0RC01PEHRR"	M 426.0	BOOL	// Pieza ejectada habilitacion de respuesta Recalage
"C0RC02PEHRR"	M 427.0	BOOL	// Pieza ejectada habilitacion de respuesta Recalage
"A11DINHIB1"	M 500.0	BOOL	// A11 DEMANDA DE MODIFICACION DE SECURIDAD
"A12DINHIB1"	M 500.1	BOOL	// A12 DEMANDA DE MODIFICACION DE SECURIDAD
"B11DINHIB1"	M 500.2	BOOL	// B11 DEMANDA DE MODIFICACION DE SECURIDAD
"B12DINHIB1"	M 500.3	BOOL	// B12 DEMANDA DE MODIFICACION DE SECURIDAD
"B13DINHIB1"	M 500.4	BOOL	// B13 DEMANDA DE MODIFICACION DE SECURIDAD
"C11DINHIB1"	M 500.5	BOOL	// C11 DEMANDA DE MODIFICACION DE SECURIDAD
"C12DINHIB1"	M 500.6	BOOL	// C12 DEMANDA DE MODIFICACION DE SECURIDAD
"C13DINHIB1"	M 500.7	BOOL	// C13 DEMANDA DE MODIFICACION DE SECURIDAD
"B21DINHIB1"	M 501.0	BOOL	// B21 DEMANDA DE MODIFICACION DE SECURIDAD
"B22DINHIB1"	M 501.1	BOOL	// B22 DEMANDA DE MODIFICACION DE SECURIDAD
"B23DINHIB1"	M 501.2	BOOL	// B23 DEMANDA DE MODIFICACION DE SECURIDAD
"C21DINHIB1"	M 501.3	BOOL	// C21 DEMANDA DE MODIFICACION DE SECURIDAD
"C22DINHIB1"	M 501.4	BOOL	// C22 DEMANDA DE MODIFICACION DE SECURIDAD
"C23DINHIB1"	M 501.5	BOOL	// C23 DEMANDA DE MODIFICACION DE SECURIDAD
"A11ACONF"	M 502.0	BOOL	// A11 AUTHORIZACION DE MODIFICACION DE SECURIDAD
"A12ACONF"	M 502.1	BOOL	// A12 AUTHORIZACION DE MODIFICACION DE SECURIDAD
"B11ACONF"	M 502.2	BOOL	// B11 AUTHORIZACION DE MODIFICACION DE SECURIDAD
"B12ACONF"	M 502.3	BOOL	// B12 AUTHORIZACION DE MODIFICACION DE SECURIDAD
"B13ACONF"	M 502.4	BOOL	// B13 AUTHORIZACION DE MODIFICACION DE SECURIDAD
"C11ACONF"	M 502.5	BOOL	// C11 AUTHORIZACION DE MODIFICACION DE SECURIDAD
"C12ACONF"	M 502.6	BOOL	// C12 AUTHORIZACION DE MODIFICACION DE SECURIDAD
"C13ACONF"	M 502.7	BOOL	// C13 AUTHORIZACION DE MODIFICACION DE SECURIDAD
"B21ACONF"	M 503.0	BOOL	// B21 AUTHORIZACION DE MODIFICACION DE SECURIDAD
"B22ACONF"	M 503.1	BOOL	// B22 AUTHORIZACION DE MODIFICACION DE SECURIDAD
"B23ACONF"	M 503.2	BOOL	// B23 AUTHORIZACION DE MODIFICACION DE SECURIDAD
"C21ACONF"	M 503.3	BOOL	// C21 AUTHORIZACION DE MODIFICACION DE SECURIDAD
"C22ACONF"	M 503.4	BOOL	// C22 AUTHORIZACION DE MODIFICACION DE SECURIDAD
"C23ACONF"	M 503.5	BOOL	// C23 AUTHORIZACION DE MODIFICACION DE SECURIDAD
"A11VINHIB"	M 504.0	BOOL	// A11 VALIDACION DE MODIFICACION DE SECURIDAD
"A12VINHIB"	M 504.1	BOOL	// A12 VALIDACION DE MODIFICACION DE SECURIDAD
"B11VINHIB"	M 504.2	BOOL	// B11 VALIDACION DE MODIFICACION DE SECURIDAD
"B12VINHIB"	M 504.3	BOOL	// B12 VALIDACION DE MODIFICACION DE SECURIDAD
"B13VINHIB"	M 504.4	BOOL	// B13 VALIDACION DE MODIFICACION DE SECURIDAD
"C11VINHIB"	M 504.5	BOOL	// C11 VALIDACION DE MODIFICACION DE SECURIDAD
"C12VINHIB"	M 504.6	BOOL	// C12 VALIDACION DE MODIFICACION DE SECURIDAD
"C13VINHIB"	M 504.7	BOOL	// C13 VALIDACION DE MODIFICACION DE SECURIDAD
"B21VINHIB"	M 505.0	BOOL	// B21 VALIDACION DE MODIFICACION DE SECURIDAD
"B22VINHIB"	M 505.1	BOOL	// B22 VALIDACION DE MODIFICACION DE SECURIDAD
"B23VINHIB"	M 505.2	BOOL	// B23 VALIDACION DE MODIFICACION DE SECURIDAD
"C21VINHIB"	M 505.3	BOOL	// C11 VALIDACION DE MODIFICACION DE SECURIDAD
"C22VINHIB"	M 505.4	BOOL	// C12 VALIDACION DE MODIFICACION DE SECURIDAD
"C23VINHIB"	M 505.5	BOOL	// C13 VALIDACION DE MODIFICACION DE SECURIDAD
"A11MINHIB"	M 506.0	BOOL	// A11 MEMORIA INHIBICION DE SECURIDAD
"A12MINHIB"	M 506.1	BOOL	// A12 MEMORIA INHIBICION DE SECURIDAD
"B11MINHIB"	M 506.2	BOOL	// B11 MEMORIA INHIBICION DE SECURIDAD
"B12MINHIB"	M 506.3	BOOL	// B12 MEMORIA INHIBICION DE SECURIDAD
"B13MINHIB"	M 506.4	BOOL	// B13 MEMORIA INHIBICION DE SECURIDAD
"C11MINHIB"	M 506.5	BOOL	// C11 MEMORIA INHIBICION DE SECURIDAD
"C12MINHIB"	M 506.6	BOOL	// C12 MEMORIA INHIBICION DE SECURIDAD
"C13MINHIB"	M 506.7	BOOL	// C13 MEMORIA INHIBICION DE SECURIDAD
"B21MINHIB"	M 507.0	BOOL	// B21 MEMORIA INHIBICION DE SECURIDAD
"B22MINHIB"	M 507.1	BOOL	// B22 MEMORIA INHIBICION DE SECURIDAD
"B23MINHIB"	M 507.2	BOOL	// B23 MEMORIA INHIBICION DE SECURIDAD
"C21MINHIB"	M 507.3	BOOL	// C11 MEMORIA INHIBICION DE SECURIDAD
"C22MINHIB"	M 507.4	BOOL	// C12 MEMORIA INHIBICION DE SECURIDAD
"C23MINHIB"	M 507.5	BOOL	// C13 MEMORIA INHIBICION DE SECURIDAD
"TSG"	M 840.0	BOOL	// Tranferecia de A0 a A0W sin guinche
"CDPRMPPB02"	MW 901	WORD	// Cantidad de Pulsos para Reset MPPB02
"CDPRMPPB01"	MW 904	WORD	// Cantidad de Pulsos para Reset MPPB01
"CDPRMPPA01"	MW 907	WORD	// Cantidad de Pulsos para Reset MPPA01
"CYCL_EXC"	OB 1	OB 1	// EXECUTION CYCLE
